KUKA KRL program: EPS_2_251112_SAMH02_A_20250918124114.src

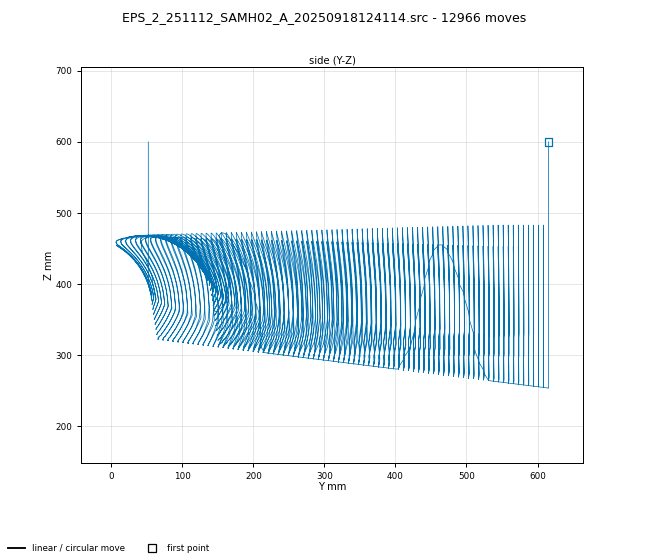
[picture p0: tool path of EPS_2_251112_SAMH02_A_20250918124114.src, 12966 of 12968 moves have a stored position in this frame; points joined in program order, loops and branches not executed]
&ACCESS RVP
&REL 4
&COMMENT QRS 19112012
&PARAM EDITMASK = *
DEF PART()
EXT BAS (BAS_COMMAND :IN,REAL :IN )
INT I
BAS (#INITMOV,0 )

;KUKA QRS Post kuka4.cps  Date:22-06-2017 !

File_ID=2849

QRS_PRE_INIT()

;Init var - Until changes are made in qrs_pre_init
Outlet_Square_prg=0
Inlet_1_Square_prg=0
Inlet_2_Square_prg=0
Inlet_3_Square_prg=0
Inlet_4_Square_prg=0
Inlet_5_Square_prg=0

Outlet_1={X 0.000, Y 541.230, Z 408.000, B 0.000, E1 0.000 }
Inlet_1={X 0.000, Y 543.360, Z 378.000, B 0.000, E1 152.000 }
Outlet_1_type=150
Inlet_1_type=150
;QRS#1=Sidecore dimensions
;QRS#2=150-6" PVC SDR 28
;QRS#3=150-6" PVC SDR 28
;QRS#4=
;QRS#5=
;QRS#6=
;QRS#7=
;QRS#8=
;QRS#9=10-06 PSX
;QRS#10=10-06 PSX
;QRS#11=
;QRS#12=
;QRS#13=
;QRS#14=
;QRS#15=
;QRS#16=1220x127x762 2,5'
;QRS#17=EPS Height
;QRS#18=483
;QRS#19=*
;QRS#20= UPDATED VERSION 22-06-2017
;QRS#21=*
Outlet_Square=070
Inlet_1_Square=070
Inlet_2_Square=0
Inlet_3_Square=0
Inlet_4_Square=0
Inlet_5_Square=0
Mill_Square=1
Outlet_Square_Prg=203
Inlet_1_Square_prg=203

QRS_INIT()

$ADVANCE=5

; T1
PTP {E1 173.623,E2 173.623}
PTP {X 0,Y 615.454,A -85,B 0,C 180,E1 173.623,E2 173.623,E3 0,E4 0,E5 0,E6 0}
QRS_SPEED_INIT()
LIN {X 0,Y 615.454,Z 600,A -85,B 0,C 180,E1 173.623,E2 173.623,E3 0,E4 0,E5 0,E6 0} C_VEL
LIN {X 0,Y 615.454,Z 263.682,A -85,B 0,C 180,E1 173.623,E2 173.623} C_VEL
LIN {X 0,Y 615.454,Z 255.505,A -85,B 0,C 180,E1 173.623,E2 173.623} C_VEL
LIN {X 0,Y 615.45,Z 253.505,A -85,B 0,C 180,E1 173.437,E2 173.437} C_VEL
LIN {X 0,Y 615.491,Z 253.512,A -85,B 0,C 180,E1 170.801,E2 170.801} C_VEL
LIN {X 0,Y 615.491,Z 253.498,A -85,B 0,C 180,E1 168.139,E2 168.139} C_VEL
LIN {X 0,Y 615.456,Z 253.5,A -85,B 0,C 180,E1 165.45,E2 165.45} C_VEL
LIN {X 0,Y 615.458,Z 253.499,A -85,B 0,C 180,E1 163.412,E2 163.412} C_VEL
LIN {X 0,Y 615.459,Z 253.499,A -85,B 0,C 180,E1 161.353,E2 161.353} C_VEL
LIN {X 0,Y 615.459,Z 253.499,A -85,B 0,C 180,E1 159.268,E2 159.268} C_VEL
LIN {X 0,Y 615.458,Z 253.5,A -85,B 0,C 180,E1 157.154,E2 157.154} C_VEL
LIN {X 0,Y 615.456,Z 253.5,A -85,B 0,C 180,E1 155.007,E2 155.007} C_VEL
LIN {X 0,Y 615.454,Z 253.502,A -85,B 0,C 180,E1 152.821,E2 152.821} C_VEL
LIN {X 0,Y 615.475,Z 253.509,A -85,B 0,C 180,E1 150.204,E2 150.204} C_VEL
LIN {X 0,Y 615.489,Z 253.502,A -85,B 0,C 180,E1 147.543,E2 147.543} C_VEL
LIN {X 0,Y 615.496,Z 253.494,A -85,B 0,C 180,E1 145.185,E2 145.185} C_VEL
LIN {X 0,Y 615.469,Z 253.497,A -85,B 0,C 180,E1 142.756,E2 142.756} C_VEL
LIN {X 0,Y 615.456,Z 253.503,A -85,B 0,C 180,E1 140.247,E2 140.247} C_VEL
LIN {X 0,Y 615.486,Z 253.511,A -85,B 0,C 180,E1 137.647,E2 137.647} C_VEL
LIN {X 0,Y 615.461,Z 253.707,A -85,B 0,C 180,E1 135.926,E2 135.926} C_VEL
LIN {X 0,Y 615.484,Z 267.327,A -85,B 0,C 180,E1 133.243,E2 133.243} C_VEL
LIN {X 0,Y 615.489,Z 280.89,A -85,B 0,C 180,E1 130.605,E2 130.605} C_VEL
LIN {X 0,Y 615.477,Z 294.187,A -85,B 0,C 180,E1 128.053,E2 128.053} C_VEL
LIN {X 0,Y 615.497,Z 369.287,A -85,B 0,C 180,E1 127.164,E2 127.164} C_VEL
LIN {X 0,Y 615.489,Z 378.589,A -85,B 0,C 180,E1 126.974,E2 126.974} C_VEL
LIN {X 0,Y 615.487,Z 386.446,A -85,B 0,C 180,E1 126.744,E2 126.744} C_VEL
LIN {X 0,Y 615.49,Z 394.748,A -85,B 0,C 180,E1 126.423,E2 126.423} C_VEL
LIN {X 0,Y 615.494,Z 402.34,A -85,B 0,C 180,E1 126.054,E2 126.054} C_VEL
LIN {X 0,Y 615.478,Z 411.206,A -85,B 0,C 180,E1 125.515,E2 125.515} C_VEL
LIN {X 0,Y 615.492,Z 419.16,A -85,B 0,C 180,E1 124.913,E2 124.913} C_VEL
LIN {X 0,Y 615.496,Z 426.942,A -85,B 0,C 180,E1 124.19,E2 124.19} C_VEL
LIN {X 0,Y 615.494,Z 433.793,A -85,B 0,C 180,E1 123.385,E2 123.385} C_VEL
LIN {X 0,Y 615.499,Z 438.844,A -85,B 0,C 180,E1 122.65,E2 122.65} C_VEL
LIN {X 0,Y 615.493,Z 442.518,A -85,B 0,C 180,E1 122.008,E2 122.008} C_VEL
LIN {X 0,Y 615.489,Z 446.578,A -85,B 0,C 180,E1 121.086,E2 121.086} C_VEL
LIN {X 0,Y 615.499,Z 449.503,A -85,B 0,C 180,E1 120.158,E2 120.158} C_VEL
LIN {X 0,Y 615.49,Z 451.13,A -85,B 0,C 180,E1 119.405,E2 119.405} C_VEL
LIN {X 0,Y 615.494,Z 452.177,A -85,B 0,C 180,E1 118.451,E2 118.451} C_VEL
LIN {X 0,Y 615.491,Z 452.386,A -85,B 0,C 180,E1 117.914,E2 117.914} C_VEL
LIN {X 0,Y 615.487,Z 451.899,A -85,B 0,C 180,E1 117.045,E2 117.045} C_VEL
LIN {X 0,Y 615.489,Z 451.043,A -85,B 0,C 180,E1 116.443,E2 116.443} C_VEL
LIN {X 0,Y 615.492,Z 449.065,A -85,B 0,C 180,E1 115.569,E2 115.569} C_VEL
LIN {X 0,Y 615.493,Z 445.858,A -85,B 0,C 180,E1 114.63,E2 114.63} C_VEL
LIN {X 0,Y 615.496,Z 441.867,A -85,B 0,C 180,E1 113.782,E2 113.782} C_VEL
LIN {X 0,Y 615.494,Z 437.323,A -85,B 0,C 180,E1 113.021,E2 113.021} C_VEL
LIN {X 0,Y 615.498,Z 430.598,A -85,B 0,C 180,E1 112.135,E2 112.135} C_VEL
LIN {X 0,Y 615.499,Z 423.976,A -85,B 0,C 180,E1 111.431,E2 111.431} C_VEL
LIN {X 0,Y 615.482,Z 415.903,A -85,B 0,C 180,E1 110.73,E2 110.73} C_VEL
LIN {X 0,Y 615.489,Z 405.501,A -85,B 0,C 180,E1 110.032,E2 110.032} C_VEL
LIN {X 0,Y 615.482,Z 397.231,A -85,B 0,C 180,E1 109.598,E2 109.598} C_VEL
LIN {X 0,Y 615.474,Z 388.91,A -85,B 0,C 180,E1 109.251,E2 109.251} C_VEL
LIN {X 0,Y 615.487,Z 379.076,A -85,B 0,C 180,E1 108.948,E2 108.948} C_VEL
LIN {X 0,Y 615.486,Z 369.76,A -85,B 0,C 180,E1 108.753,E2 108.753} C_VEL
LIN {X 0,Y 615.48,Z 294.091,A -85,B 0,C 180,E1 107.849,E2 107.849} C_VEL
LIN {X 0,Y 615.493,Z 280.475,A -85,B 0,C 180,E1 105.225,E2 105.225} C_VEL
LIN {X 0,Y 615.475,Z 266.63,A -85,B 0,C 180,E1 102.53,E2 102.53} C_VEL
LIN {X 0,Y 615.472,Z 253.502,A -85,B 0,C 180,E1 99.924,E2 99.924} C_VEL
LIN {X 0,Y 615.484,Z 253.494,A -85,B 0,C 180,E1 97.215,E2 97.215} C_VEL
LIN {X 0,Y 615.48,Z 253.504,A -85,B 0,C 180,E1 94.584,E2 94.584} C_VEL
LIN {X 0,Y 615.483,Z 253.509,A -85,B 0,C 180,E1 91.963,E2 91.963} C_VEL
LIN {X 0,Y 615.472,Z 253.498,A -85,B 0,C 180,E1 89.346,E2 89.346} C_VEL
LIN {X 0,Y 615.489,Z 253.494,A -85,B 0,C 180,E1 86.727,E2 86.727} C_VEL
LIN {X 0,Y 615.485,Z 253.507,A -85,B 0,C 180,E1 84.102,E2 84.102} C_VEL
LIN {X 0,Y 615.475,Z 253.506,A -85,B 0,C 180,E1 81.463,E2 81.463} C_VEL
LIN {X 0,Y 615.479,Z 253.495,A -85,B 0,C 180,E1 78.807,E2 78.807} C_VEL
LIN {X 0,Y 615.48,Z 253.501,A -85,B 0,C 180,E1 76.071,E2 76.071} C_VEL
LIN {X 0,Y 615.484,Z 253.513,A -85,B 0,C 180,E1 73.414,E2 73.414} C_VEL
LIN {X 0,Y 615.469,Z 253.498,A -85,B 0,C 180,E1 70.662,E2 70.662} C_VEL
LIN {X 0,Y 615.484,Z 253.498,A -85,B 0,C 180,E1 67.864,E2 67.864} C_VEL
LIN {X 0,Y 615.481,Z 253.509,A -85,B 0,C 180,E1 65.009,E2 65.009} C_VEL
LIN {X 0,Y 615.474,Z 253.507,A -85,B 0,C 180,E1 62.823,E2 62.823} C_VEL
LIN {X 0,Y 615.47,Z 253.497,A -85,B 0,C 180,E1 60.209,E2 60.209} C_VEL
LIN {X 0,Y 615.488,Z 253.496,A -85,B 0,C 180,E1 57.544,E2 57.544} C_VEL
LIN {X 0,Y 615.484,Z 253.504,A -85,B 0,C 180,E1 55.186,E2 55.186} C_VEL
LIN {X 0,Y 615.49,Z 253.515,A -85,B 0,C 180,E1 52.759,E2 52.759} C_VEL
LIN {X 0,Y 615.464,Z 253.499,A -85,B 0,C 180,E1 49.914,E2 49.914} C_VEL
LIN {X 0,Y 615.472,Z 253.496,A -85,B 0,C 180,E1 47.647,E2 47.647} C_VEL
LIN {X 0,Y 615.486,Z 253.5,A -85,B 0,C 180,E1 44.933,E2 44.933} C_VEL
LIN {X 0,Y 615.494,Z 253.512,A -85,B 0,C 180,E1 42.353,E2 42.353} C_VEL
LIN {X 0,Y 615.461,Z 253.503,A -85,B 0,C 180,E1 39.752,E2 39.752} C_VEL
LIN {X 0,Y 615.486,Z 253.495,A -85,B 0,C 180,E1 36.939,E2 36.939} C_VEL
LIN {X 0,Y 615.491,Z 253.511,A -85,B 0,C 180,E1 34.022,E2 34.022} C_VEL
LIN {X 0,Y 615.468,Z 253.507,A -85,B 0,C 180,E1 31.687,E2 31.687} C_VEL
LIN {X 0,Y 615.459,Z 253.504,A -85,B 0,C 180,E1 29.408,E2 29.408} C_VEL
LIN {X 0,Y 615.46,Z 253.5,A -85,B 0,C 180,E1 27.043,E2 27.043} C_VEL
LIN {X 0,Y 615.491,Z 253.497,A -85,B 0,C 180,E1 24.272,E2 24.272} C_VEL
LIN {X 0,Y 615.476,Z 253.509,A -85,B 0,C 180,E1 21.432,E2 21.432} C_VEL
LIN {X 0,Y 615.474,Z 253.509,A -85,B 0,C 180,E1 19.338,E2 19.338} C_VEL
LIN {X 0,Y 615.46,Z 253.499,A -85,B 0,C 180,E1 16.587,E2 16.587} C_VEL
LIN {X 0,Y 615.492,Z 253.498,A -85,B 0,C 180,E1 13.874,E2 13.874} C_VEL
LIN {X 0,Y 615.486,Z 253.511,A -85,B 0,C 180,E1 11.193,E2 11.193} C_VEL
LIN {X 0,Y 615.452,Z 253.503,A -85,B 0,C 180,E1 8.537,E2 8.537} C_VEL
LIN {X 0,Y 615.48,Z 253.495,A -85,B 0,C 180,E1 5.899,E2 5.899} C_VEL
LIN {X 0,Y 615.491,Z 253.504,A -85,B 0,C 180,E1 3.273,E2 3.273} C_VEL
LIN {X 0,Y 615.47,Z 253.509,A -85,B 0,C 180,E1 0.654,E2 0.654} C_VEL
LIN {X 0,Y 615.451,Z 253.502,A -85,B 0,C 180,E1 -1.963,E2 -1.963} C_VEL
LIN {X 0,Y 615.488,Z 253.495,A -85,B 0,C 180,E1 -4.584,E2 -4.584} C_VEL
LIN {X 0,Y 615.489,Z 253.509,A -85,B 0,C 180,E1 -7.216,E2 -7.216} C_VEL
LIN {X 0,Y 615.458,Z 253.507,A -85,B 0,C 180,E1 -9.863,E2 -9.863} C_VEL
LIN {X 0,Y 615.463,Z 253.508,A -85,B 0,C 180,E1 -11.861,E2 -11.861} C_VEL
LIN {X 0,Y 615.463,Z 253.508,A -85,B 0,C 180,E1 -13.93,E2 -13.93} C_VEL
LIN {X 0,Y 615.447,Z 253.503,A -85,B 0,C 180,E1 -16.424,E2 -16.424} C_VEL
LIN {X 0,Y 615.449,Z 253.502,A -85,B 0,C 180,E1 -18.647,E2 -18.647} C_VEL
LIN {X 0,Y 615.494,Z 253.499,A -85,B 0,C 180,E1 -21.432,E2 -21.432} C_VEL
LIN {X 0,Y 615.464,Z 253.509,A -85,B 0,C 180,E1 -24.273,E2 -24.273} C_VEL
LIN {X 0,Y 615.456,Z 253.508,A -85,B 0,C 180,E1 -26.446,E2 -26.446} C_VEL
LIN {X 0,Y 615.447,Z 253.507,A -85,B 0,C 180,E1 -28.66,E2 -28.66} C_VEL
LIN {X 0,Y 615.444,Z 253.503,A -85,B 0,C 180,E1 -31.082,E2 -31.082} C_VEL
LIN {X 0,Y 615.467,Z 253.499,A -85,B 0,C 180,E1 -33.534,E2 -33.534} C_VEL
LIN {X 0,Y 615.482,Z 253.515,A -85,B 0,C 180,E1 -36.425,E2 -36.425} C_VEL
LIN {X 0,Y 615.445,Z 253.507,A -85,B 0,C 180,E1 -39.059,E2 -39.059} C_VEL
LIN {X 0,Y 615.44,Z 253.504,A -85,B 0,C 180,E1 -41.478,E2 -41.478} C_VEL
LIN {X 0,Y 615.49,Z 253.497,A -85,B 0,C 180,E1 -44.149,E2 -44.149} C_VEL
LIN {X 0,Y 615.475,Z 253.511,A -85,B 0,C 180,E1 -46.954,E2 -46.954} C_VEL
LIN {X 0,Y 615.445,Z 253.507,A -85,B 0,C 180,E1 -49.392,E2 -49.392} C_VEL
LIN {X 0,Y 615.441,Z 253.503,A -85,B 0,C 180,E1 -51.929,E2 -51.929} C_VEL
LIN {X 0,Y 615.469,Z 253.5,A -85,B 0,C 180,E1 -54.384,E2 -54.384} C_VEL
LIN {X 0,Y 615.491,Z 253.501,A -85,B 0,C 180,E1 -56.765,E2 -56.765} C_VEL
LIN {X 0,Y 615.497,Z 253.508,A -85,B 0,C 180,E1 -59.082,E2 -59.082} C_VEL
LIN {X 0,Y 615.464,Z 253.51,A -85,B 0,C 180,E1 -61.554,E2 -61.554} C_VEL
LIN {X 0,Y 615.47,Z 253.511,A -85,B 0,C 180,E1 -63.556,E2 -63.556} C_VEL
LIN {X 0,Y 615.441,Z 253.508,A -85,B 0,C 180,E1 -66.001,E2 -66.001} C_VEL
LIN {X 0,Y 615.455,Z 253.51,A -85,B 0,C 180,E1 -67.863,E2 -67.863} C_VEL
LIN {X 0,Y 615.467,Z 253.526,A -85,B 0,C 180,E1 -68.963,E2 -68.963} C_VEL
LIN {X 0,Y 615.453,Z 271.669,A -85,B 0,C 180,E1 -71.881,E2 -71.881} C_VEL
LIN {X 0,Y 615.482,Z 287.773,A -85,B 0,C 180,E1 -74.435,E2 -74.435} C_VEL
LIN {X 0,Y 615.47,Z 305.003,A -85,B 0,C 180,E1 -77.135,E2 -77.135} C_VEL
LIN {X 0,Y 615.485,Z 322.619,A -85,B 0,C 180,E1 -79.868,E2 -79.868} C_VEL
LIN {X 0,Y 615.472,Z 399.961,A -85,B 0,C 180,E1 -80.801,E2 -80.801} C_VEL
LIN {X 0,Y 615.465,Z 409.713,A -85,B 0,C 180,E1 -81.008,E2 -81.008} C_VEL
LIN {X 0,Y 615.472,Z 420.166,A -85,B 0,C 180,E1 -81.339,E2 -81.339} C_VEL
LIN {X 0,Y 615.498,Z 430.431,A -85,B 0,C 180,E1 -81.794,E2 -81.794} C_VEL
LIN {X 0,Y 615.477,Z 440.204,A -85,B 0,C 180,E1 -82.372,E2 -82.372} C_VEL
LIN {X 0,Y 615.493,Z 447.937,A -85,B 0,C 180,E1 -82.942,E2 -82.942} C_VEL
LIN {X 0,Y 615.497,Z 455.336,A -85,B 0,C 180,E1 -83.608,E2 -83.608} C_VEL
LIN {X 0,Y 615.498,Z 462.739,A -85,B 0,C 180,E1 -84.43,E2 -84.43} C_VEL
LIN {X 0,Y 615.497,Z 468.533,A -85,B 0,C 180,E1 -85.252,E2 -85.252} C_VEL
LIN {X 0,Y 615.494,Z 473.101,A -85,B 0,C 180,E1 -86.072,E2 -86.072} C_VEL
LIN {X 0,Y 615.493,Z 476.069,A -85,B 0,C 180,E1 -86.727,E2 -86.727} C_VEL
LIN {X 0,Y 615.494,Z 478.357,A -85,B 0,C 180,E1 -87.382,E2 -87.382} C_VEL
LIN {X 0,Y 615.499,Z 480.085,A -85,B 0,C 180,E1 -88.037,E2 -88.037} C_VEL
LIN {X 0,Y 615.493,Z 481.33,A -85,B 0,C 180,E1 -88.691,E2 -88.691} C_VEL
LIN {X 0,Y 615.491,Z 482.104,A -85,B 0,C 180,E1 -89.346,E2 -89.346} C_VEL
LIN {X 0,Y 615.491,Z 482.389,A -85,B 0,C 180,E1 -90,E2 -90} C_VEL
LIN {X 0,Y 615.491,Z 482.104,A -85,B 0,C 180,E1 -90.654,E2 -90.654} C_VEL
LIN {X 0,Y 615.493,Z 481.33,A -85,B 0,C 180,E1 -91.309,E2 -91.309} C_VEL
LIN {X 0,Y 615.499,Z 480.085,A -85,B 0,C 180,E1 -91.963,E2 -91.963} C_VEL
LIN {X 0,Y 615.488,Z 477.221,A -85,B 0,C 180,E1 -92.945,E2 -92.945} C_VEL
LIN {X 0,Y 615.492,Z 474.604,A -85,B 0,C 180,E1 -93.601,E2 -93.601} C_VEL
LIN {X 0,Y 615.497,Z 469.483,A -85,B 0,C 180,E1 -94.584,E2 -94.584} C_VEL
LIN {X 0,Y 615.495,Z 463.969,A -85,B 0,C 180,E1 -95.405,E2 -95.405} C_VEL
LIN {X 0,Y 615.498,Z 457.02,A -85,B 0,C 180,E1 -96.227,E2 -96.227} C_VEL
LIN {X 0,Y 615.495,Z 449.86,A -85,B 0,C 180,E1 -96.901,E2 -96.901} C_VEL
LIN {X 0,Y 615.477,Z 442.628,A -85,B 0,C 180,E1 -97.463,E2 -97.463} C_VEL
LIN {X 0,Y 615.495,Z 434.873,A -85,B 0,C 180,E1 -97.958,E2 -97.958} C_VEL
LIN {X 0,Y 615.494,Z 426.92,A -85,B 0,C 180,E1 -98.371,E2 -98.371} C_VEL
LIN {X 0,Y 615.468,Z 417.771,A -85,B 0,C 180,E1 -98.743,E2 -98.743} C_VEL
LIN {X 0,Y 615.465,Z 409.714,A -85,B 0,C 180,E1 -98.992,E2 -98.992} C_VEL
LIN {X 0,Y 615.472,Z 399.963,A -85,B 0,C 180,E1 -99.199,E2 -99.199} C_VEL
LIN {X 0,Y 615.482,Z 322.62,A -85,B 0,C 180,E1 -100.132,E2 -100.132} C_VEL
LIN {X 0,Y 615.47,Z 305.003,A -85,B 0,C 180,E1 -102.865,E2 -102.865} C_VEL
LIN {X 0,Y 615.482,Z 287.773,A -85,B 0,C 180,E1 -105.565,E2 -105.565} C_VEL
LIN {X 0,Y 615.459,Z 270.657,A -85,B 0,C 180,E1 -108.28,E2 -108.28} C_VEL
LIN {X 0,Y 615.464,Z 253.501,A -85,B 0,C 180,E1 -111.059,E2 -111.059} C_VEL
LIN {X 0,Y 615.437,Z 253.504,A -85,B 0,C 180,E1 -113.558,E2 -113.558} C_VEL
LIN {X 0,Y 615.435,Z 253.505,A -85,B 0,C 180,E1 -115.717,E2 -115.717} C_VEL
LIN {X 0,Y 615.435,Z 253.506,A -85,B 0,C 180,E1 -117.917,E2 -117.917} C_VEL
LIN {X 0,Y 615.437,Z 253.507,A -85,B 0,C 180,E1 -120.162,E2 -120.162} C_VEL
LIN {X 0,Y 615.451,Z 253.509,A -85,B 0,C 180,E1 -122.458,E2 -122.458} C_VEL
LIN {X 0,Y 615.48,Z 253.512,A -85,B 0,C 180,E1 -124.814,E2 -124.814} C_VEL
LIN {X 0,Y 615.496,Z 253.505,A -85,B 0,C 180,E1 -127.24,E2 -127.24} C_VEL
LIN {X 0,Y 615.472,Z 253.499,A -85,B 0,C 180,E1 -129.75,E2 -129.75} C_VEL
LIN {X 0,Y 615.439,Z 253.504,A -85,B 0,C 180,E1 -132.356,E2 -132.356} C_VEL
LIN {X 0,Y 615.455,Z 253.509,A -85,B 0,C 180,E1 -134.928,E2 -134.928} C_VEL
LIN {X 0,Y 615.494,Z 253.505,A -85,B 0,C 180,E1 -137.648,E2 -137.648} C_VEL
LIN {X 0,Y 615.462,Z 253.5,A -85,B 0,C 180,E1 -140.248,E2 -140.248} C_VEL
LIN {X 0,Y 615.441,Z 253.504,A -85,B 0,C 180,E1 -142.755,E2 -142.755} C_VEL
LIN {X 0,Y 615.455,Z 253.509,A -85,B 0,C 180,E1 -145.301,E2 -145.301} C_VEL
LIN {X 0,Y 615.485,Z 253.511,A -85,B 0,C 180,E1 -147.667,E2 -147.667} C_VEL
LIN {X 0,Y 615.47,Z 253.499,A -85,B 0,C 180,E1 -150.593,E2 -150.593} C_VEL
LIN {X 0,Y 615.447,Z 253.502,A -85,B 0,C 180,E1 -152.959,E2 -152.959} C_VEL
LIN {X 0,Y 615.451,Z 253.501,A -85,B 0,C 180,E1 -155.007,E2 -155.007} C_VEL
LIN {X 0,Y 615.448,Z 253.502,A -85,B 0,C 180,E1 -157.154,E2 -157.154} C_VEL
LIN {X 0,Y 615.444,Z 253.504,A -85,B 0,C 180,E1 -159.449,E2 -159.449} C_VEL
LIN {X 0,Y 615.469,Z 253.51,A -85,B 0,C 180,E1 -162.043,E2 -162.043} C_VEL
LIN {X 0,Y 615.495,Z 253.5,A -85,B 0,C 180,E1 -164.774,E2 -164.774} C_VEL
LIN {X 0,Y 615.453,Z 253.5,A -85,B 0,C 180,E1 -167.469,E2 -167.469} C_VEL
LIN {X 0,Y 615.458,Z 253.499,A -85,B 0,C 180,E1 -169.473,E2 -169.473} C_VEL
LIN {X 0,Y 615.466,Z 253.498,A -85,B 0,C 180,E1 -171.463,E2 -171.463} C_VEL
LIN {X 0,Y 615.448,Z 253.505,A -85,B 0,C 180,E1 -174.101,E2 -174.101} C_VEL
LIN {X 0,Y 615.486,Z 253.512,A -85,B 0,C 180,E1 -176.727,E2 -176.727} C_VEL
LIN {X 0,Y 615.49,Z 253.499,A -85,B 0,C 180,E1 -179.346,E2 -179.346} C_VEL
LIN {X 0,Y 615.459,Z 253.499,A -85,B 0,C 180,E1 -181.963,E2 -181.963} C_VEL
LIN {X 0,Y 615.453,Z 253.506,A -85,B 0,C 180,E1 -184.585,E2 -184.585} C_VEL
LIN {X 0,Y 615.45,Z 253.505,A -85,B 0,C 180,E1 -186.563,E2 -186.563} C_VEL
LIN {X 0,Y 614.799,Z 253.659,A -85,B 0,C 180,E1 -187.109,E2 -187.109} C_VEL
LIN {X 0,Y 611.984,Z 254.059,A -85,B 0,C 180,E1 -187.996,E2 -187.996} C_VEL
LIN {X 0,Y 609.593,Z 254.377,A -85,B 0,C 180,E1 -188.708,E2 -188.708} C_VEL
LIN {X 0,Y 608.554,Z 254.498,A -85,B 0,C 180,E1 -189.258,E2 -189.258} C_VEL
LIN {X 0,Y 608.463,Z 254.506,A -85,B 0,C 180,E1 -189.444,E2 -189.444} C_VEL
LIN {X 0,Y 608.457,Z 254.5,A -85,B 0,C 180,E1 -192,E2 -192} C_VEL
LIN {X 0,Y 608.45,Z 254.5,A -85,B 0,C 180,E1 -194.721,E2 -194.721} C_VEL
LIN {X 0,Y 608.422,Z 254.503,A -85,B 0,C 180,E1 -196.785,E2 -196.785} C_VEL
LIN {X 0,Y 608.441,Z 254.511,A -85,B 0,C 180,E1 -199.571,E2 -199.571} C_VEL
LIN {X 0,Y 608.45,Z 254.5,A -85,B 0,C 180,E1 -202.478,E2 -202.478} C_VEL
LIN {X 0,Y 608.443,Z 254.501,A -85,B 0,C 180,E1 -204.572,E2 -204.572} C_VEL
LIN {X 0,Y 608.451,Z 254.5,A -85,B 0,C 180,E1 -207.206,E2 -207.206} C_VEL
LIN {X 0,Y 608.462,Z 254.509,A -85,B 0,C 180,E1 -209.974,E2 -209.974} C_VEL
LIN {X 0,Y 608.445,Z 254.5,A -85,B 0,C 180,E1 -212.88,E2 -212.88} C_VEL
LIN {X 0,Y 608.43,Z 254.501,A -85,B 0,C 180,E1 -215.279,E2 -215.279} C_VEL
LIN {X 0,Y 608.453,Z 254.501,A -85,B 0,C 180,E1 -217.748,E2 -217.748} C_VEL
LIN {X 0,Y 608.444,Z 254.511,A -85,B 0,C 180,E1 -220.33,E2 -220.33} C_VEL
LIN {X 0,Y 608.477,Z 254.496,A -85,B 0,C 180,E1 -223.311,E2 -223.311} C_VEL
LIN {X 0,Y 608.445,Z 254.617,A -85,B 0,C 180,E1 -224.02,E2 -224.02} C_VEL
LIN {X 0,Y 608.471,Z 268.075,A -85,B 0,C 180,E1 -226.691,E2 -226.691} C_VEL
LIN {X 0,Y 608.441,Z 282.321,A -85,B 0,C 180,E1 -229.48,E2 -229.48} C_VEL
LIN {X 0,Y 608.437,Z 294.377,A -85,B 0,C 180,E1 -231.818,E2 -231.818} C_VEL
LIN {X 0,Y 608.509,Z 369.385,A -85,B 0,C 180,E1 -232.723,E2 -232.723} C_VEL
LIN {X 0,Y 608.501,Z 378.797,A -85,B 0,C 180,E1 -232.917,E2 -232.917} C_VEL
LIN {X 0,Y 608.505,Z 387.885,A -85,B 0,C 180,E1 -233.193,E2 -233.193} C_VEL
LIN {X 0,Y 608.487,Z 396.712,A -85,B 0,C 180,E1 -233.553,E2 -233.553} C_VEL
LIN {X 0,Y 608.479,Z 405.514,A -85,B 0,C 180,E1 -234.012,E2 -234.012} C_VEL
LIN {X 0,Y 608.446,Z 414.814,A -85,B 0,C 180,E1 -234.622,E2 -234.622} C_VEL
LIN {X 0,Y 608.45,Z 423.03,A -85,B 0,C 180,E1 -235.313,E2 -235.313} C_VEL
LIN {X 0,Y 608.467,Z 429.1,A -85,B 0,C 180,E1 -235.931,E2 -235.931} C_VEL
LIN {X 0,Y 608.436,Z 435.483,A -85,B 0,C 180,E1 -236.725,E2 -236.725} C_VEL
LIN {X 0,Y 608.433,Z 440.417,A -85,B 0,C 180,E1 -237.482,E2 -237.482} C_VEL
LIN {X 0,Y 608.427,Z 444.651,A -85,B 0,C 180,E1 -238.294,E2 -238.294} C_VEL
LIN {X 0,Y 608.421,Z 447.88,A -85,B 0,C 180,E1 -239.093,E2 -239.093} C_VEL
LIN {X 0,Y 608.425,Z 450.622,A -85,B 0,C 180,E1 -240.036,E2 -240.036} C_VEL
LIN {X 0,Y 608.409,Z 452.298,A -85,B 0,C 180,E1 -240.978,E2 -240.978} C_VEL
LIN {X 0,Y 608.438,Z 452.878,A -85,B 0,C 180,E1 -241.734,E2 -241.734} C_VEL
LIN {X 0,Y 608.429,Z 452.666,A -85,B 0,C 180,E1 -242.802,E2 -242.802} C_VEL
LIN {X 0,Y 608.417,Z 450.84,A -85,B 0,C 180,E1 -243.964,E2 -243.964} C_VEL
LIN {X 0,Y 608.429,Z 447.648,A -85,B 0,C 180,E1 -245.064,E2 -245.064} C_VEL
LIN {X 0,Y 608.426,Z 444.364,A -85,B 0,C 180,E1 -245.859,E2 -245.859} C_VEL
LIN {X 0,Y 608.431,Z 439.909,A -85,B 0,C 180,E1 -246.696,E2 -246.696} C_VEL
LIN {X 0,Y 608.458,Z 433.846,A -85,B 0,C 180,E1 -247.595,E2 -247.595} C_VEL
LIN {X 0,Y 608.467,Z 425.99,A -85,B 0,C 180,E1 -248.487,E2 -248.487} C_VEL
LIN {X 0,Y 608.454,Z 419.135,A -85,B 0,C 180,E1 -249.117,E2 -249.117} C_VEL
LIN {X 0,Y 608.457,Z 412.982,A -85,B 0,C 180,E1 -249.594,E2 -249.594} C_VEL
LIN {X 0,Y 608.464,Z 405.503,A -85,B 0,C 180,E1 -250.079,E2 -250.079} C_VEL
LIN {X 0,Y 608.465,Z 397.14,A -85,B 0,C 180,E1 -250.518,E2 -250.518} C_VEL
LIN {X 0,Y 608.488,Z 388.671,A -85,B 0,C 180,E1 -250.87,E2 -250.87} C_VEL
LIN {X 0,Y 608.508,Z 378.997,A -85,B 0,C 180,E1 -251.168,E2 -251.168} C_VEL
LIN {X 0,Y 608.506,Z 369.825,A -85,B 0,C 180,E1 -251.36,E2 -251.36} C_VEL
LIN {X 0,Y 608.447,Z 294.455,A -85,B 0,C 180,E1 -252.263,E2 -252.263} C_VEL
LIN {X 0,Y 608.442,Z 280.641,A -85,B 0,C 180,E1 -254.937,E2 -254.937} C_VEL
LIN {X 0,Y 608.477,Z 268.457,A -85,B 0,C 180,E1 -257.324,E2 -257.324} C_VEL
LIN {X 0,Y 608.468,Z 254.532,A -85,B 0,C 180,E1 -260.086,E2 -260.086} C_VEL
LIN {X 0,Y 608.463,Z 254.497,A -85,B 0,C 180,E1 -262.701,E2 -262.701} C_VEL
LIN {X 0,Y 608.45,Z 254.504,A -85,B 0,C 180,E1 -265.362,E2 -265.362} C_VEL
LIN {X 0,Y 608.453,Z 254.507,A -85,B 0,C 180,E1 -268.014,E2 -268.014} C_VEL
LIN {X 0,Y 608.468,Z 254.498,A -85,B 0,C 180,E1 -270.662,E2 -270.662} C_VEL
LIN {X 0,Y 608.482,Z 254.496,A -85,B 0,C 180,E1 -273.311,E2 -273.311} C_VEL
LIN {X 0,Y 608.457,Z 254.507,A -85,B 0,C 180,E1 -275.967,E2 -275.967} C_VEL
LIN {X 0,Y 608.448,Z 254.503,A -85,B 0,C 180,E1 -278.636,E2 -278.636} C_VEL
LIN {X 0,Y 608.456,Z 254.498,A -85,B 0,C 180,E1 -281.324,E2 -281.324} C_VEL
LIN {X 0,Y 608.47,Z 254.501,A -85,B 0,C 180,E1 -284.037,E2 -284.037} C_VEL
LIN {X 0,Y 608.455,Z 254.505,A -85,B 0,C 180,E1 -286.783,E2 -286.783} C_VEL
LIN {X 0,Y 608.442,Z 254.5,A -85,B 0,C 180,E1 -289.57,E2 -289.57} C_VEL
LIN {X 0,Y 608.477,Z 254.502,A -85,B 0,C 180,E1 -292.405,E2 -292.405} C_VEL
LIN {X 0,Y 608.45,Z 254.507,A -85,B 0,C 180,E1 -294.57,E2 -294.57} C_VEL
LIN {X 0,Y 608.471,Z 254.502,A -85,B 0,C 180,E1 -297.206,E2 -297.206} C_VEL
LIN {X 0,Y 608.461,Z 254.498,A -85,B 0,C 180,E1 -299.97,E2 -299.97} C_VEL
LIN {X 0,Y 608.454,Z 254.506,A -85,B 0,C 180,E1 -302.879,E2 -302.879} C_VEL
LIN {X 0,Y 608.432,Z 254.511,A -85,B 0,C 180,E1 -305.277,E2 -305.277} C_VEL
LIN {X 0,Y 608.457,Z 254.501,A -85,B 0,C 180,E1 -307.746,E2 -307.746} C_VEL
LIN {X 0,Y 608.442,Z 254.5,A -85,B 0,C 180,E1 -310.328,E2 -310.328} C_VEL
LIN {X 0,Y 608.474,Z 254.505,A -85,B 0,C 180,E1 -313.309,E2 -313.309} C_VEL
LIN {X 0,Y 608.454,Z 254.501,A -85,B 0,C 180,E1 -316.129,E2 -316.129} C_VEL
LIN {X 0,Y 608.452,Z 254.499,A -85,B 0,C 180,E1 -318.823,E2 -318.823} C_VEL
LIN {X 0,Y 608.463,Z 254.509,A -85,B 0,C 180,E1 -321.758,E2 -321.758} C_VEL
LIN {X 0,Y 608.466,Z 254.506,A -85,B 0,C 180,E1 -323.95,E2 -323.95} C_VEL
LIN {X 0,Y 608.435,Z 254.505,A -85,B 0,C 180,E1 -326.327,E2 -326.327} C_VEL
LIN {X 0,Y 608.432,Z 254.502,A -85,B 0,C 180,E1 -328.732,E2 -328.732} C_VEL
LIN {X 0,Y 608.471,Z 254.497,A -85,B 0,C 180,E1 -331.377,E2 -331.377} C_VEL
LIN {X 0,Y 608.467,Z 254.507,A -85,B 0,C 180,E1 -334.276,E2 -334.276} C_VEL
LIN {X 0,Y 608.434,Z 254.503,A -85,B 0,C 180,E1 -336.875,E2 -336.875} C_VEL
LIN {X 0,Y 608.451,Z 254.499,A -85,B 0,C 180,E1 -339.321,E2 -339.321} C_VEL
LIN {X 0,Y 608.442,Z 254.502,A -85,B 0,C 180,E1 -341.828,E2 -341.828} C_VEL
LIN {X 0,Y 608.464,Z 254.509,A -85,B 0,C 180,E1 -344.594,E2 -344.594} C_VEL
LIN {X 0,Y 608.452,Z 254.5,A -85,B 0,C 180,E1 -347.322,E2 -347.322} C_VEL
LIN {X 0,Y 608.457,Z 254.499,A -85,B 0,C 180,E1 -350.023,E2 -350.023} C_VEL
LIN {X 0,Y 608.479,Z 254.504,A -85,B 0,C 180,E1 -352.701,E2 -352.701} C_VEL
LIN {X 0,Y 608.428,Z 254.506,A -85,B 0,C 180,E1 -355.362,E2 -355.362} C_VEL
LIN {X 0,Y 608.455,Z 254.504,A -85,B 0,C 180,E1 -357.352,E2 -357.352} C_VEL
LIN {X 0,Y 608.447,Z 254.499,A -85,B 0,C 180,E1 -360,E2 -360} C_VEL
LIN {X 0,Y 608.482,Z 254.497,A -85,B 0,C 180,E1 -362.648,E2 -362.648} C_VEL
LIN {X 0,Y 608.471,Z 254.508,A -85,B 0,C 180,E1 -365.302,E2 -365.302} C_VEL
LIN {X 0,Y 608.45,Z 254.501,A -85,B 0,C 180,E1 -367.967,E2 -367.967} C_VEL
LIN {X 0,Y 608.447,Z 254.5,A -85,B 0,C 180,E1 -370.65,E2 -370.65} C_VEL
LIN {X 0,Y 608.462,Z 254.505,A -85,B 0,C 180,E1 -373.356,E2 -373.356} C_VEL
LIN {X 0,Y 608.437,Z 254.505,A -85,B 0,C 180,E1 -376.094,E2 -376.094} C_VEL
LIN {X 0,Y 608.436,Z 254.501,A -85,B 0,C 180,E1 -378.87,E2 -378.87} C_VEL
LIN {X 0,Y 608.466,Z 254.505,A -85,B 0,C 180,E1 -381.692,E2 -381.692} C_VEL
LIN {X 0,Y 608.428,Z 254.504,A -85,B 0,C 180,E1 -384.572,E2 -384.572} C_VEL
LIN {X 0,Y 608.451,Z 254.499,A -85,B 0,C 180,E1 -387.206,E2 -387.206} C_VEL
LIN {X 0,Y 608.474,Z 254.504,A -85,B 0,C 180,E1 -389.976,E2 -389.976} C_VEL
LIN {X 0,Y 608.433,Z 254.503,A -85,B 0,C 180,E1 -392.881,E2 -392.881} C_VEL
LIN {X 0,Y 608.417,Z 254.503,A -85,B 0,C 180,E1 -395.279,E2 -395.279} C_VEL
LIN {X 0,Y 608.455,Z 254.499,A -85,B 0,C 180,E1 -397.747,E2 -397.747} C_VEL
LIN {X 0,Y 608.473,Z 254.504,A -85,B 0,C 180,E1 -400.333,E2 -400.333} C_VEL
LIN {X 0,Y 608.425,Z 254.508,A -85,B 0,C 180,E1 -402.962,E2 -402.962} C_VEL
LIN {X 0,Y 608.427,Z 254.505,A -85,B 0,C 180,E1 -405.203,E2 -405.203} C_VEL
LIN {X 0,Y 608.436,Z 254.507,A -85,B 0,C 180,E1 -407.04,E2 -407.04} C_VEL
LIN {X 0,Y 608.41,Z 254.504,A -85,B 0,C 180,E1 -409.695,E2 -409.695} C_VEL
LIN {X 0,Y 608.445,Z 254.501,A -85,B 0,C 180,E1 -412.253,E2 -412.253} C_VEL
LIN {X 0,Y 608.445,Z 254.511,A -85,B 0,C 180,E1 -415.095,E2 -415.095} C_VEL
LIN {X 0,Y 608.428,Z 254.502,A -85,B 0,C 180,E1 -417.904,E2 -417.904} C_VEL
LIN {X 0,Y 608.423,Z 254.502,A -85,B 0,C 180,E1 -420.219,E2 -420.219} C_VEL
LIN {X 0,Y 608.458,Z 254.501,A -85,B 0,C 180,E1 -422.797,E2 -422.797} C_VEL
LIN {X 0,Y 608.445,Z 254.504,A -85,B 0,C 180,E1 -425.854,E2 -425.854} C_VEL
LIN {X 0,Y 608.429,Z 254.503,A -85,B 0,C 180,E1 -428.308,E2 -428.308} C_VEL
LIN {X 0,Y 608.456,Z 254.629,A -85,B 0,C 180,E1 -428.886,E2 -428.886} C_VEL
LIN {X 0,Y 608.48,Z 271.013,A -85,B 0,C 180,E1 -431.551,E2 -431.551} C_VEL
LIN {X 0,Y 608.5,Z 287.882,A -85,B 0,C 180,E1 -434.252,E2 -434.252} C_VEL
LIN {X 0,Y 608.443,Z 305.184,A -85,B 0,C 180,E1 -436.983,E2 -436.983} C_VEL
LIN {X 0,Y 608.471,Z 322.892,A -85,B 0,C 180,E1 -439.75,E2 -439.75} C_VEL
LIN {X 0,Y 608.495,Z 400.46,A -85,B 0,C 180,E1 -440.695,E2 -440.695} C_VEL
LIN {X 0,Y 608.464,Z 410.085,A -85,B 0,C 180,E1 -440.904,E2 -440.904} C_VEL
LIN {X 0,Y 608.479,Z 421.623,A -85,B 0,C 180,E1 -441.281,E2 -441.281} C_VEL
LIN {X 0,Y 608.479,Z 432.237,A -85,B 0,C 180,E1 -441.783,E2 -441.783} C_VEL
LIN {X 0,Y 608.458,Z 440.545,A -85,B 0,C 180,E1 -442.284,E2 -442.284} C_VEL
LIN {X 0,Y 608.459,Z 448.403,A -85,B 0,C 180,E1 -442.868,E2 -442.868} C_VEL
LIN {X 0,Y 608.466,Z 455.358,A -85,B 0,C 180,E1 -443.496,E2 -443.496} C_VEL
LIN {X 0,Y 608.469,Z 463.192,A -85,B 0,C 180,E1 -444.366,E2 -444.366} C_VEL
LIN {X 0,Y 608.448,Z 469.028,A -85,B 0,C 180,E1 -445.196,E2 -445.196} C_VEL
LIN {X 0,Y 608.432,Z 473.631,A -85,B 0,C 180,E1 -446.026,E2 -446.026} C_VEL
LIN {X 0,Y 608.425,Z 476.622,A -85,B 0,C 180,E1 -446.689,E2 -446.689} C_VEL
LIN {X 0,Y 608.423,Z 478.931,A -85,B 0,C 180,E1 -447.352,E2 -447.352} C_VEL
LIN {X 0,Y 608.443,Z 480.678,A -85,B 0,C 180,E1 -448.014,E2 -448.014} C_VEL
LIN {X 0,Y 608.446,Z 481.934,A -85,B 0,C 180,E1 -448.676,E2 -448.676} C_VEL
LIN {X 0,Y 608.434,Z 482.714,A -85,B 0,C 180,E1 -449.338,E2 -449.338} C_VEL
LIN {X 0,Y 608.431,Z 483,A -85,B 0,C 180,E1 -450,E2 -450} C_VEL
LIN {X 0,Y 608.434,Z 482.714,A -85,B 0,C 180,E1 -450.662,E2 -450.662} C_VEL
LIN {X 0,Y 608.446,Z 481.934,A -85,B 0,C 180,E1 -451.324,E2 -451.324} C_VEL
LIN {X 0,Y 608.443,Z 480.678,A -85,B 0,C 180,E1 -451.986,E2 -451.986} C_VEL
LIN {X 0,Y 608.444,Z 477.786,A -85,B 0,C 180,E1 -452.979,E2 -452.979} C_VEL
LIN {X 0,Y 608.446,Z 475.147,A -85,B 0,C 180,E1 -453.642,E2 -453.642} C_VEL
LIN {X 0,Y 608.447,Z 469.986,A -85,B 0,C 180,E1 -454.638,E2 -454.638} C_VEL
LIN {X 0,Y 608.46,Z 464.431,A -85,B 0,C 180,E1 -455.468,E2 -455.468} C_VEL
LIN {X 0,Y 608.455,Z 456.67,A -85,B 0,C 180,E1 -456.376,E2 -456.376} C_VEL
LIN {X 0,Y 608.452,Z 449.418,A -85,B 0,C 180,E1 -457.049,E2 -457.049} C_VEL
LIN {X 0,Y 608.458,Z 441.763,A -85,B 0,C 180,E1 -457.633,E2 -457.633} C_VEL
LIN {X 0,Y 608.497,Z 433.724,A -85,B 0,C 180,E1 -458.134,E2 -458.134} C_VEL
LIN {X 0,Y 608.483,Z 425.395,A -85,B 0,C 180,E1 -458.552,E2 -458.552} C_VEL
LIN {X 0,Y 608.459,Z 416.896,A -85,B 0,C 180,E1 -458.887,E2 -458.887} C_VEL
LIN {X 0,Y 608.491,Z 407.596,A -85,B 0,C 180,E1 -459.159,E2 -459.159} C_VEL
LIN {X 0,Y 608.483,Z 397.864,A -85,B 0,C 180,E1 -459.347,E2 -459.347} C_VEL
LIN {X 0,Y 608.449,Z 322.892,A -85,B 0,C 180,E1 -460.25,E2 -460.25} C_VEL
LIN {X 0,Y 608.443,Z 304.103,A -85,B 0,C 180,E1 -463.186,E2 -463.186} C_VEL
LIN {X 0,Y 608.492,Z 286.8,A -85,B 0,C 180,E1 -465.92,E2 -465.92} C_VEL
LIN {X 0,Y 608.51,Z 269.285,A -85,B 0,C 180,E1 -468.727,E2 -468.727} C_VEL
LIN {X 0,Y 608.428,Z 254.504,A -85,B 0,C 180,E1 -471.137,E2 -471.137} C_VEL
LIN {X 0,Y 608.433,Z 254.503,A -85,B 0,C 180,E1 -473.124,E2 -473.124} C_VEL
LIN {X 0,Y 608.431,Z 254.501,A -85,B 0,C 180,E1 -475.713,E2 -475.713} C_VEL
LIN {X 0,Y 608.416,Z 254.507,A -85,B 0,C 180,E1 -478.267,E2 -478.267} C_VEL
LIN {X 0,Y 608.436,Z 254.508,A -85,B 0,C 180,E1 -480.546,E2 -480.546} C_VEL
LIN {X 0,Y 608.447,Z 254.512,A -85,B 0,C 180,E1 -482.879,E2 -482.879} C_VEL
LIN {X 0,Y 608.431,Z 254.507,A -85,B 0,C 180,E1 -485.277,E2 -485.277} C_VEL
LIN {X 0,Y 608.445,Z 254.501,A -85,B 0,C 180,E1 -487.747,E2 -487.747} C_VEL
LIN {X 0,Y 608.424,Z 254.503,A -85,B 0,C 180,E1 -490.326,E2 -490.326} C_VEL
LIN {X 0,Y 608.435,Z 254.507,A -85,B 0,C 180,E1 -492.96,E2 -492.96} C_VEL
LIN {X 0,Y 608.456,Z 254.503,A -85,B 0,C 180,E1 -495.734,E2 -495.734} C_VEL
LIN {X 0,Y 608.471,Z 254.499,A -85,B 0,C 180,E1 -497.94,E2 -497.94} C_VEL
LIN {X 0,Y 608.415,Z 254.503,A -85,B 0,C 180,E1 -500.556,E2 -500.556} C_VEL
LIN {X 0,Y 608.418,Z 254.506,A -85,B 0,C 180,E1 -503.082,E2 -503.082} C_VEL
LIN {X 0,Y 608.451,Z 254.507,A -85,B 0,C 180,E1 -505.53,E2 -505.53} C_VEL
LIN {X 0,Y 608.465,Z 254.507,A -85,B 0,C 180,E1 -507.906,E2 -507.906} C_VEL
LIN {X 0,Y 608.477,Z 254.501,A -85,B 0,C 180,E1 -510.221,E2 -510.221} C_VEL
LIN {X 0,Y 608.45,Z 254.499,A -85,B 0,C 180,E1 -512.795,E2 -512.795} C_VEL
LIN {X 0,Y 608.426,Z 254.504,A -85,B 0,C 180,E1 -515.428,E2 -515.428} C_VEL
LIN {X 0,Y 608.464,Z 254.506,A -85,B 0,C 180,E1 -518.308,E2 -518.308} C_VEL
LIN {X 0,Y 608.441,Z 254.5,A -85,B 0,C 180,E1 -521.287,E2 -521.287} C_VEL
LIN {X 0,Y 608.434,Z 254.505,A -85,B 0,C 180,E1 -523.906,E2 -523.906} C_VEL
LIN {X 0,Y 608.461,Z 254.506,A -85,B 0,C 180,E1 -526.644,E2 -526.644} C_VEL
LIN {X 0,Y 608.446,Z 254.5,A -85,B 0,C 180,E1 -529.35,E2 -529.35} C_VEL
LIN {X 0,Y 608.447,Z 254.501,A -85,B 0,C 180,E1 -532.033,E2 -532.033} C_VEL
LIN {X 0,Y 608.468,Z 254.508,A -85,B 0,C 180,E1 -534.698,E2 -534.698} C_VEL
LIN {X 0,Y 608.482,Z 254.498,A -85,B 0,C 180,E1 -537.352,E2 -537.352} C_VEL
LIN {X 0,Y 608.445,Z 254.499,A -85,B 0,C 180,E1 -540,E2 -540} C_VEL
LIN {X 0,Y 608.451,Z 254.503,A -85,B 0,C 180,E1 -542.648,E2 -542.648} C_VEL
LIN {X 0,Y 608.468,Z 254.505,A -85,B 0,C 180,E1 -545.302,E2 -545.302} C_VEL
LIN {X 0,Y 608.468,Z 254.497,A -85,B 0,C 180,E1 -547.967,E2 -547.967} C_VEL
LIN {X 0,Y 608.463,Z 254.506,A -85,B 0,C 180,E1 -549.444,E2 -549.444} C_VEL
LIN {X 0,Y 607.781,Z 254.585,A -85,B 0,C 180,E1 -549.997,E2 -549.997} C_VEL
LIN {X 0,Y 604.925,Z 254.942,A -85,B 0,C 180,E1 -550.893,E2 -550.893} C_VEL
LIN {X 0,Y 602.52,Z 255.244,A -85,B 0,C 180,E1 -551.615,E2 -551.615} C_VEL
LIN {X 0,Y 601.483,Z 255.368,A -85,B 0,C 180,E1 -552.171,E2 -552.171} C_VEL
LIN {X 0,Y 601.395,Z 255.377,A -85,B 0,C 180,E1 -552.36,E2 -552.36} C_VEL
LIN {X 0,Y 601.41,Z 255.378,A -85,B 0,C 180,E1 -554.898,E2 -554.898} C_VEL
LIN {X 0,Y 601.397,Z 255.38,A -85,B 0,C 180,E1 -556.987,E2 -556.987} C_VEL
LIN {X 0,Y 601.397,Z 255.386,A -85,B 0,C 180,E1 -559.81,E2 -559.81} C_VEL
LIN {X 0,Y 601.399,Z 255.378,A -85,B 0,C 180,E1 -562.684,E2 -562.684} C_VEL
LIN {X 0,Y 601.387,Z 255.379,A -85,B 0,C 180,E1 -564.879,E2 -564.879} C_VEL
LIN {X 0,Y 601.395,Z 255.38,A -85,B 0,C 180,E1 -567.362,E2 -567.362} C_VEL
LIN {X 0,Y 601.437,Z 255.382,A -85,B 0,C 180,E1 -570.164,E2 -570.164} C_VEL
LIN {X 0,Y 601.416,Z 255.377,A -85,B 0,C 180,E1 -572.717,E2 -572.717} C_VEL
LIN {X 0,Y 601.406,Z 255.376,A -85,B 0,C 180,E1 -575.116,E2 -575.116} C_VEL
LIN {X 0,Y 601.424,Z 255.375,A -85,B 0,C 180,E1 -577.42,E2 -577.42} C_VEL
LIN {X 0,Y 601.4,Z 255.382,A -85,B 0,C 180,E1 -579.996,E2 -579.996} C_VEL
LIN {X 0,Y 601.408,Z 255.385,A -85,B 0,C 180,E1 -582.671,E2 -582.671} C_VEL
LIN {X 0,Y 601.425,Z 255.557,A -85,B 0,C 180,E1 -583.992,E2 -583.992} C_VEL
LIN {X 0,Y 601.428,Z 268.824,A -85,B 0,C 180,E1 -586.656,E2 -586.656} C_VEL
LIN {X 0,Y 601.394,Z 282.821,A -85,B 0,C 180,E1 -589.429,E2 -589.429} C_VEL
LIN {X 0,Y 601.377,Z 294.376,A -85,B 0,C 180,E1 -591.696,E2 -591.696} C_VEL
LIN {X 0,Y 601.507,Z 369.143,A -85,B 0,C 180,E1 -592.609,E2 -592.609} C_VEL
LIN {X 0,Y 601.479,Z 378.784,A -85,B 0,C 180,E1 -592.809,E2 -592.809} C_VEL
LIN {X 0,Y 601.476,Z 388.492,A -85,B 0,C 180,E1 -593.11,E2 -593.11} C_VEL
LIN {X 0,Y 601.458,Z 398.068,A -85,B 0,C 180,E1 -593.515,E2 -593.515} C_VEL
LIN {X 0,Y 601.41,Z 409.396,A -85,B 0,C 180,E1 -594.158,E2 -594.158} C_VEL
LIN {X 0,Y 601.395,Z 417.689,A -85,B 0,C 180,E1 -594.769,E2 -594.769} C_VEL
LIN {X 0,Y 601.412,Z 424.455,A -85,B 0,C 180,E1 -595.375,E2 -595.375} C_VEL
LIN {X 0,Y 601.376,Z 430.908,A -85,B 0,C 180,E1 -596.073,E2 -596.073} C_VEL
LIN {X 0,Y 601.372,Z 436.793,A -85,B 0,C 180,E1 -596.85,E2 -596.85} C_VEL
LIN {X 0,Y 601.344,Z 442.938,A -85,B 0,C 180,E1 -597.876,E2 -597.876} C_VEL
LIN {X 0,Y 601.35,Z 446.036,A -85,B 0,C 180,E1 -598.557,E2 -598.557} C_VEL
LIN {X 0,Y 601.352,Z 449.198,A -85,B 0,C 180,E1 -599.445,E2 -599.445} C_VEL
LIN {X 0,Y 601.336,Z 451.791,A -85,B 0,C 180,E1 -600.603,E2 -600.603} C_VEL
LIN {X 0,Y 601.325,Z 452.71,A -85,B 0,C 180,E1 -601.369,E2 -601.369} C_VEL
LIN {X 0,Y 601.332,Z 452.984,A -85,B 0,C 180,E1 -602.129,E2 -602.129} C_VEL
LIN {X 0,Y 601.326,Z 452.61,A -85,B 0,C 180,E1 -602.884,E2 -602.884} C_VEL
LIN {X 0,Y 601.311,Z 451.583,A -85,B 0,C 180,E1 -603.633,E2 -603.633} C_VEL
LIN {X 0,Y 601.335,Z 448.846,A -85,B 0,C 180,E1 -604.75,E2 -604.75} C_VEL
LIN {X 0,Y 601.325,Z 445.143,A -85,B 0,C 180,E1 -605.731,E2 -605.731} C_VEL
LIN {X 0,Y 601.363,Z 441.878,A -85,B 0,C 180,E1 -606.406,E2 -606.406} C_VEL
LIN {X 0,Y 601.36,Z 437.536,A -85,B 0,C 180,E1 -607.134,E2 -607.134} C_VEL
LIN {X 0,Y 601.373,Z 432.23,A -85,B 0,C 180,E1 -607.861,E2 -607.861} C_VEL
LIN {X 0,Y 601.412,Z 425.799,A -85,B 0,C 180,E1 -608.582,E2 -608.582} C_VEL
LIN {X 0,Y 601.4,Z 418.107,A -85,B 0,C 180,E1 -609.286,E2 -609.286} C_VEL
LIN {X 0,Y 601.418,Z 410.79,A -85,B 0,C 180,E1 -609.835,E2 -609.835} C_VEL
LIN {X 0,Y 601.427,Z 402.057,A -85,B 0,C 180,E1 -610.37,E2 -610.37} C_VEL
LIN {X 0,Y 601.479,Z 390.647,A -85,B 0,C 180,E1 -610.904,E2 -610.904} C_VEL
LIN {X 0,Y 601.49,Z 379.692,A -85,B 0,C 180,E1 -611.258,E2 -611.258} C_VEL
LIN {X 0,Y 601.511,Z 370.659,A -85,B 0,C 180,E1 -611.456,E2 -611.456} C_VEL
LIN {X 0,Y 601.499,Z 327.876,A -85,B 0,C 180,E1 -611.986,E2 -611.986} C_VEL
LIN {X 0,Y 601.417,Z 294.916,A -85,B 0,C 180,E1 -612.379,E2 -612.379} C_VEL
LIN {X 0,Y 601.387,Z 294.344,A -85,B 0,C 180,E1 -612.4,E2 -612.4} C_VEL
LIN {X 0,Y 601.373,Z 280.585,A -85,B 0,C 180,E1 -615.102,E2 -615.102} C_VEL
LIN {X 0,Y 601.433,Z 268.413,A -85,B 0,C 180,E1 -617.516,E2 -617.516} C_VEL
LIN {X 0,Y 601.415,Z 255.379,A -85,B 0,C 180,E1 -620.16,E2 -620.16} C_VEL
LIN {X 0,Y 601.44,Z 255.372,A -85,B 0,C 180,E1 -622.615,E2 -622.615} C_VEL
LIN {X 0,Y 601.419,Z 255.379,A -85,B 0,C 180,E1 -625.308,E2 -625.308} C_VEL
LIN {X 0,Y 601.423,Z 255.383,A -85,B 0,C 180,E1 -627.991,E2 -627.991} C_VEL
LIN {X 0,Y 601.441,Z 255.373,A -85,B 0,C 180,E1 -630.67,E2 -630.67} C_VEL
LIN {X 0,Y 601.433,Z 255.374,A -85,B 0,C 180,E1 -633.349,E2 -633.349} C_VEL
LIN {X 0,Y 601.407,Z 255.386,A -85,B 0,C 180,E1 -636.037,E2 -636.037} C_VEL
LIN {X 0,Y 601.437,Z 255.382,A -85,B 0,C 180,E1 -638.061,E2 -638.061} C_VEL
LIN {X 0,Y 601.42,Z 255.376,A -85,B 0,C 180,E1 -641.009,E2 -641.009} C_VEL
LIN {X 0,Y 601.411,Z 255.376,A -85,B 0,C 180,E1 -643.516,E2 -643.516} C_VEL
LIN {X 0,Y 601.439,Z 255.38,A -85,B 0,C 180,E1 -646.286,E2 -646.286} C_VEL
LIN {X 0,Y 601.415,Z 255.378,A -85,B 0,C 180,E1 -649.098,E2 -649.098} C_VEL
LIN {X 0,Y 601.402,Z 255.379,A -85,B 0,C 180,E1 -651.239,E2 -651.239} C_VEL
LIN {X 0,Y 601.458,Z 255.372,A -85,B 0,C 180,E1 -654.14,E2 -654.14} C_VEL
LIN {X 0,Y 601.445,Z 255.379,A -85,B 0,C 180,E1 -657.111,E2 -657.111} C_VEL
LIN {X 0,Y 601.409,Z 255.38,A -85,B 0,C 180,E1 -659.393,E2 -659.393} C_VEL
LIN {X 0,Y 601.399,Z 255.379,A -85,B 0,C 180,E1 -661.726,E2 -661.726} C_VEL
LIN {X 0,Y 601.415,Z 255.375,A -85,B 0,C 180,E1 -664.118,E2 -664.118} C_VEL
LIN {X 0,Y 601.432,Z 255.382,A -85,B 0,C 180,E1 -667.381,E2 -667.381} C_VEL
LIN {X 0,Y 601.395,Z 255.379,A -85,B 0,C 180,E1 -669.995,E2 -669.995} C_VEL
LIN {X 0,Y 601.405,Z 255.377,A -85,B 0,C 180,E1 -672.669,E2 -672.669} C_VEL
LIN {X 0,Y 601.419,Z 255.386,A -85,B 0,C 180,E1 -675.481,E2 -675.481} C_VEL
LIN {X 0,Y 601.414,Z 255.376,A -85,B 0,C 180,E1 -678.406,E2 -678.406} C_VEL
LIN {X 0,Y 601.43,Z 255.374,A -85,B 0,C 180,E1 -680.875,E2 -680.875} C_VEL
LIN {X 0,Y 601.435,Z 255.383,A -85,B 0,C 180,E1 -683.733,E2 -683.733} C_VEL
LIN {X 0,Y 601.423,Z 255.383,A -85,B 0,C 180,E1 -686.063,E2 -686.063} C_VEL
LIN {X 0,Y 601.407,Z 255.379,A -85,B 0,C 180,E1 -688.545,E2 -688.545} C_VEL
LIN {X 0,Y 601.432,Z 255.373,A -85,B 0,C 180,E1 -691.209,E2 -691.209} C_VEL
LIN {X 0,Y 601.398,Z 255.38,A -85,B 0,C 180,E1 -693.636,E2 -693.636} C_VEL
LIN {X 0,Y 601.41,Z 255.382,A -85,B 0,C 180,E1 -696.589,E2 -696.589} C_VEL
LIN {X 0,Y 601.419,Z 255.375,A -85,B 0,C 180,E1 -699.478,E2 -699.478} C_VEL
LIN {X 0,Y 601.389,Z 255.387,A -85,B 0,C 180,E1 -702.311,E2 -702.311} C_VEL
LIN {X 0,Y 601.414,Z 255.384,A -85,B 0,C 180,E1 -704.409,E2 -704.409} C_VEL
LIN {X 0,Y 601.402,Z 255.38,A -85,B 0,C 180,E1 -707.171,E2 -707.171} C_VEL
LIN {X 0,Y 601.428,Z 255.374,A -85,B 0,C 180,E1 -709.905,E2 -709.905} C_VEL
LIN {X 0,Y 601.446,Z 255.379,A -85,B 0,C 180,E1 -712.615,E2 -712.615} C_VEL
LIN {X 0,Y 601.4,Z 255.382,A -85,B 0,C 180,E1 -715.308,E2 -715.308} C_VEL
LIN {X 0,Y 601.402,Z 255.377,A -85,B 0,C 180,E1 -717.991,E2 -717.991} C_VEL
LIN {X 0,Y 601.451,Z 255.374,A -85,B 0,C 180,E1 -720.669,E2 -720.669} C_VEL
LIN {X 0,Y 601.425,Z 255.383,A -85,B 0,C 180,E1 -723.349,E2 -723.349} C_VEL
LIN {X 0,Y 601.383,Z 255.38,A -85,B 0,C 180,E1 -726.037,E2 -726.037} C_VEL
LIN {X 0,Y 601.416,Z 255.377,A -85,B 0,C 180,E1 -728.061,E2 -728.061} C_VEL
LIN {X 0,Y 601.459,Z 255.373,A -85,B 0,C 180,E1 -731.038,E2 -731.038} C_VEL
LIN {X 0,Y 601.404,Z 255.38,A -85,B 0,C 180,E1 -734.092,E2 -734.092} C_VEL
LIN {X 0,Y 601.401,Z 255.378,A -85,B 0,C 180,E1 -736.987,E2 -736.987} C_VEL
LIN {X 0,Y 601.396,Z 255.39,A -85,B 0,C 180,E1 -739.81,E2 -739.81} C_VEL
LIN {X 0,Y 601.397,Z 255.378,A -85,B 0,C 180,E1 -742.684,E2 -742.684} C_VEL
LIN {X 0,Y 601.384,Z 255.379,A -85,B 0,C 180,E1 -744.879,E2 -744.879} C_VEL
LIN {X 0,Y 601.408,Z 255.384,A -85,B 0,C 180,E1 -747.868,E2 -747.868} C_VEL
LIN {X 0,Y 601.437,Z 255.385,A -85,B 0,C 180,E1 -750.163,E2 -750.163} C_VEL
LIN {X 0,Y 601.41,Z 255.376,A -85,B 0,C 180,E1 -753.315,E2 -753.315} C_VEL
LIN {X 0,Y 601.432,Z 255.383,A -85,B 0,C 180,E1 -756.267,E2 -756.267} C_VEL
LIN {X 0,Y 601.386,Z 255.381,A -85,B 0,C 180,E1 -759.128,E2 -759.128} C_VEL
LIN {X 0,Y 601.413,Z 255.376,A -85,B 0,C 180,E1 -761.766,E2 -761.766} C_VEL
LIN {X 0,Y 601.416,Z 255.384,A -85,B 0,C 180,E1 -764.536,E2 -764.536} C_VEL
LIN {X 0,Y 601.442,Z 255.378,A -85,B 0,C 180,E1 -766.426,E2 -766.426} C_VEL
LIN {X 0,Y 601.398,Z 255.38,A -85,B 0,C 180,E1 -769.429,E2 -769.429} C_VEL
LIN {X 0,Y 601.385,Z 255.38,A -85,B 0,C 180,E1 -771.731,E2 -771.731} C_VEL
LIN {X 0,Y 601.372,Z 255.381,A -85,B 0,C 180,E1 -774.246,E2 -774.246} C_VEL
LIN {X 0,Y 601.408,Z 255.38,A -85,B 0,C 180,E1 -776.686,E2 -776.686} C_VEL
LIN {X 0,Y 601.4,Z 255.386,A -85,B 0,C 180,E1 -779.058,E2 -779.058} C_VEL
LIN {X 0,Y 601.423,Z 255.385,A -85,B 0,C 180,E1 -781.374,E2 -781.374} C_VEL
LIN {X 0,Y 601.388,Z 255.385,A -85,B 0,C 180,E1 -783.636,E2 -783.636} C_VEL
LIN {X 0,Y 601.425,Z 255.378,A -85,B 0,C 180,E1 -785.859,E2 -785.859} C_VEL
LIN {X 0,Y 601.416,Z 255.44,A -85,B 0,C 180,E1 -788.762,E2 -788.762} C_VEL
LIN {X 0,Y 601.524,Z 268.416,A -85,B 0,C 180,E1 -790.905,E2 -790.905} C_VEL
LIN {X 0,Y 601.456,Z 285.719,A -85,B 0,C 180,E1 -793.714,E2 -793.714} C_VEL
LIN {X 0,Y 601.403,Z 301.187,A -85,B 0,C 180,E1 -796.192,E2 -796.192} C_VEL
LIN {X 0,Y 601.401,Z 317.877,A -85,B 0,C 180,E1 -798.838,E2 -798.838} C_VEL
LIN {X 0,Y 601.407,Z 322.892,A -85,B 0,C 180,E1 -799.628,E2 -799.628} C_VEL
LIN {X 0,Y 601.524,Z 387.927,A -85,B 0,C 180,E1 -800.416,E2 -800.416} C_VEL
LIN {X 0,Y 601.491,Z 404.182,A -85,B 0,C 180,E1 -800.649,E2 -800.649} C_VEL
LIN {X 0,Y 601.457,Z 415.693,A -85,B 0,C 180,E1 -800.967,E2 -800.967} C_VEL
LIN {X 0,Y 601.468,Z 423.542,A -85,B 0,C 180,E1 -801.263,E2 -801.263} C_VEL
LIN {X 0,Y 601.448,Z 432.24,A -85,B 0,C 180,E1 -801.686,E2 -801.686} C_VEL
LIN {X 0,Y 601.402,Z 440.547,A -85,B 0,C 180,E1 -802.192,E2 -802.192} C_VEL
LIN {X 0,Y 601.409,Z 448.404,A -85,B 0,C 180,E1 -802.783,E2 -802.783} C_VEL
LIN {X 0,Y 601.411,Z 455.598,A -85,B 0,C 180,E1 -803.443,E2 -803.443} C_VEL
LIN {X 0,Y 601.391,Z 463.192,A -85,B 0,C 180,E1 -804.299,E2 -804.299} C_VEL
LIN {X 0,Y 601.38,Z 469.028,A -85,B 0,C 180,E1 -805.14,E2 -805.14} C_VEL
LIN {X 0,Y 601.344,Z 473.631,A -85,B 0,C 180,E1 -805.979,E2 -805.979} C_VEL
LIN {X 0,Y 601.344,Z 476.622,A -85,B 0,C 180,E1 -806.65,E2 -806.65} C_VEL
LIN {X 0,Y 601.326,Z 478.932,A -85,B 0,C 180,E1 -807.321,E2 -807.321} C_VEL
LIN {X 0,Y 601.342,Z 480.679,A -85,B 0,C 180,E1 -807.991,E2 -807.991} C_VEL
LIN {X 0,Y 601.345,Z 481.934,A -85,B 0,C 180,E1 -808.661,E2 -808.661} C_VEL
LIN {X 0,Y 601.335,Z 482.713,A -85,B 0,C 180,E1 -809.33,E2 -809.33} C_VEL
LIN {X 0,Y 601.332,Z 483,A -85,B 0,C 180,E1 -810,E2 -810} C_VEL
LIN {X 0,Y 601.335,Z 482.713,A -85,B 0,C 180,E1 -810.67,E2 -810.67} C_VEL
LIN {X 0,Y 601.345,Z 481.934,A -85,B 0,C 180,E1 -811.339,E2 -811.339} C_VEL
LIN {X 0,Y 601.342,Z 480.679,A -85,B 0,C 180,E1 -812.009,E2 -812.009} C_VEL
LIN {X 0,Y 601.343,Z 477.787,A -85,B 0,C 180,E1 -813.015,E2 -813.015} C_VEL
LIN {X 0,Y 601.364,Z 475.147,A -85,B 0,C 180,E1 -813.685,E2 -813.685} C_VEL
LIN {X 0,Y 601.366,Z 469.986,A -85,B 0,C 180,E1 -814.692,E2 -814.692} C_VEL
LIN {X 0,Y 601.383,Z 464.431,A -85,B 0,C 180,E1 -815.532,E2 -815.532} C_VEL
LIN {X 0,Y 601.393,Z 457.152,A -85,B 0,C 180,E1 -816.403,E2 -816.403} C_VEL
LIN {X 0,Y 601.413,Z 449.419,A -85,B 0,C 180,E1 -817.132,E2 -817.132} C_VEL
LIN {X 0,Y 601.424,Z 441.766,A -85,B 0,C 180,E1 -817.723,E2 -817.723} C_VEL
LIN {X 0,Y 601.454,Z 433.727,A -85,B 0,C 180,E1 -818.229,E2 -818.229} C_VEL
LIN {X 0,Y 601.451,Z 425.398,A -85,B 0,C 180,E1 -818.652,E2 -818.652} C_VEL
LIN {X 0,Y 601.446,Z 416.898,A -85,B 0,C 180,E1 -818.991,E2 -818.991} C_VEL
LIN {X 0,Y 601.47,Z 406.766,A -85,B 0,C 180,E1 -819.288,E2 -819.288} C_VEL
LIN {X 0,Y 601.504,Z 395.084,A -85,B 0,C 180,E1 -819.499,E2 -819.499} C_VEL
LIN {X 0,Y 601.454,Z 323.538,A -85,B 0,C 180,E1 -820.349,E2 -820.349} C_VEL
LIN {X 0,Y 601.406,Z 322.757,A -85,B 0,C 180,E1 -820.393,E2 -820.393} C_VEL
LIN {X 0,Y 601.396,Z 304.103,A -85,B 0,C 180,E1 -823.344,E2 -823.344} C_VEL
LIN {X 0,Y 601.482,Z 287.882,A -85,B 0,C 180,E1 -825.937,E2 -825.937} C_VEL
LIN {X 0,Y 601.523,Z 269.923,A -85,B 0,C 180,E1 -828.848,E2 -828.848} C_VEL
LIN {X 0,Y 601.555,Z 256.967,A -85,B 0,C 180,E1 -830.98,E2 -830.98} C_VEL
LIN {X 0,Y 601.387,Z 255.383,A -85,B 0,C 180,E1 -831.284,E2 -831.284} C_VEL
LIN {X 0,Y 601.425,Z 255.379,A -85,B 0,C 180,E1 -834.141,E2 -834.141} C_VEL
LIN {X 0,Y 601.435,Z 255.377,A -85,B 0,C 180,E1 -837.111,E2 -837.111} C_VEL
LIN {X 0,Y 601.393,Z 255.38,A -85,B 0,C 180,E1 -839.394,E2 -839.394} C_VEL
LIN {X 0,Y 601.382,Z 255.38,A -85,B 0,C 180,E1 -841.727,E2 -841.727} C_VEL
LIN {X 0,Y 601.406,Z 255.377,A -85,B 0,C 180,E1 -844.119,E2 -844.119} C_VEL
LIN {X 0,Y 601.431,Z 255.379,A -85,B 0,C 180,E1 -847.381,E2 -847.381} C_VEL
LIN {X 0,Y 601.382,Z 255.38,A -85,B 0,C 180,E1 -849.996,E2 -849.996} C_VEL
LIN {X 0,Y 601.37,Z 255.383,A -85,B 0,C 180,E1 -852.672,E2 -852.672} C_VEL
LIN {X 0,Y 601.388,Z 255.38,A -85,B 0,C 180,E1 -854.532,E2 -854.532} C_VEL
LIN {X 0,Y 601.405,Z 255.389,A -85,B 0,C 180,E1 -857.408,E2 -857.408} C_VEL
LIN {X 0,Y 601.397,Z 255.381,A -85,B 0,C 180,E1 -860.004,E2 -860.004} C_VEL
LIN {X 0,Y 601.417,Z 255.375,A -85,B 0,C 180,E1 -862.618,E2 -862.618} C_VEL
LIN {X 0,Y 601.378,Z 255.382,A -85,B 0,C 180,E1 -865.066,E2 -865.066} C_VEL
LIN {X 0,Y 601.415,Z 255.382,A -85,B 0,C 180,E1 -867.483,E2 -867.483} C_VEL
LIN {X 0,Y 601.438,Z 255.385,A -85,B 0,C 180,E1 -869.847,E2 -869.847} C_VEL
LIN {X 0,Y 601.403,Z 255.376,A -85,B 0,C 180,E1 -872.887,E2 -872.887} C_VEL
LIN {X 0,Y 601.383,Z 255.379,A -85,B 0,C 180,E1 -875.121,E2 -875.121} C_VEL
LIN {X 0,Y 601.4,Z 255.378,A -85,B 0,C 180,E1 -877.394,E2 -877.394} C_VEL
LIN {X 0,Y 601.395,Z 255.389,A -85,B 0,C 180,E1 -880.19,E2 -880.19} C_VEL
LIN {X 0,Y 601.4,Z 255.378,A -85,B 0,C 180,E1 -883.013,E2 -883.013} C_VEL
LIN {X 0,Y 601.394,Z 255.379,A -85,B 0,C 180,E1 -885.794,E2 -885.794} C_VEL
LIN {X 0,Y 601.424,Z 255.386,A -85,B 0,C 180,E1 -888.542,E2 -888.542} C_VEL
LIN {X 0,Y 601.423,Z 255.376,A -85,B 0,C 180,E1 -891.262,E2 -891.262} C_VEL
LIN {X 0,Y 601.439,Z 255.374,A -85,B 0,C 180,E1 -893.324,E2 -893.324} C_VEL
LIN {X 0,Y 601.373,Z 255.381,A -85,B 0,C 180,E1 -895.979,E2 -895.979} C_VEL
LIN {X 0,Y 601.393,Z 255.378,A -85,B 0,C 180,E1 -897.991,E2 -897.991} C_VEL
LIN {X 0,Y 601.415,Z 255.375,A -85,B 0,C 180,E1 -900,E2 -900} C_VEL
LIN {X 0,Y 601.419,Z 255.379,A -85,B 0,C 180,E1 -902.679,E2 -902.679} C_VEL
LIN {X 0,Y 601.431,Z 255.38,A -85,B 0,C 180,E1 -905.364,E2 -905.364} C_VEL
LIN {X 0,Y 601.428,Z 255.374,A -85,B 0,C 180,E1 -908.061,E2 -908.061} C_VEL
LIN {X 0,Y 601.388,Z 255.381,A -85,B 0,C 180,E1 -910.777,E2 -910.777} C_VEL
LIN {X 0,Y 601.395,Z 255.377,A -85,B 0,C 180,E1 -912.36,E2 -912.36} C_VEL
LIN {X 0,Y 600.722,Z 255.466,A -85,B 0,C 180,E1 -912.919,E2 -912.919} C_VEL
LIN {X 0,Y 597.868,Z 255.822,A -85,B 0,C 180,E1 -913.827,E2 -913.827} C_VEL
LIN {X 0,Y 595.464,Z 256.121,A -85,B 0,C 180,E1 -914.557,E2 -914.557} C_VEL
LIN {X 0,Y 594.434,Z 256.25,A -85,B 0,C 180,E1 -915.121,E2 -915.121} C_VEL
LIN {X 0,Y 594.351,Z 256.259,A -85,B 0,C 180,E1 -915.311,E2 -915.311} C_VEL
LIN {X 0,Y 594.366,Z 256.259,A -85,B 0,C 180,E1 -917.905,E2 -917.905} C_VEL
LIN {X 0,Y 594.362,Z 256.255,A -85,B 0,C 180,E1 -920.917,E2 -920.917} C_VEL
LIN {X 0,Y 594.383,Z 256.262,A -85,B 0,C 180,E1 -923.704,E2 -923.704} C_VEL
LIN {X 0,Y 594.37,Z 256.253,A -85,B 0,C 180,E1 -926.7,E2 -926.7} C_VEL
LIN {X 0,Y 594.371,Z 256.253,A -85,B 0,C 180,E1 -928.999,E2 -928.999} C_VEL
LIN {X 0,Y 594.365,Z 256.257,A -85,B 0,C 180,E1 -931.644,E2 -931.644} C_VEL
LIN {X 0,Y 594.391,Z 256.255,A -85,B 0,C 180,E1 -934.579,E2 -934.579} C_VEL
LIN {X 0,Y 594.378,Z 256.253,A -85,B 0,C 180,E1 -937.087,E2 -937.087} C_VEL
LIN {X 0,Y 594.363,Z 256.256,A -85,B 0,C 180,E1 -939.775,E2 -939.775} C_VEL
LIN {X 0,Y 594.363,Z 256.264,A -85,B 0,C 180,E1 -942.376,E2 -942.376} C_VEL
LIN {X 0,Y 594.379,Z 256.457,A -85,B 0,C 180,E1 -943.955,E2 -943.955} C_VEL
LIN {X 0,Y 594.398,Z 268.645,A -85,B 0,C 180,E1 -946.434,E2 -946.434} C_VEL
LIN {X 0,Y 594.338,Z 282.348,A -85,B 0,C 180,E1 -949.183,E2 -949.183} C_VEL
LIN {X 0,Y 594.31,Z 294.353,A -85,B 0,C 180,E1 -951.567,E2 -951.567} C_VEL
LIN {X 0,Y 594.543,Z 303.676,A -85,B 0,C 180,E1 -951.696,E2 -951.696} C_VEL
LIN {X 0,Y 594.52,Z 369.72,A -85,B 0,C 180,E1 -952.507,E2 -952.507} C_VEL
LIN {X 0,Y 594.493,Z 379.111,A -85,B 0,C 180,E1 -952.708,E2 -952.708} C_VEL
LIN {X 0,Y 594.473,Z 388.46,A -85,B 0,C 180,E1 -953.003,E2 -953.003} C_VEL
LIN {X 0,Y 594.45,Z 399.06,A -85,B 0,C 180,E1 -953.459,E2 -953.459} C_VEL
LIN {X 0,Y 594.364,Z 409.514,A -85,B 0,C 180,E1 -954.072,E2 -954.072} C_VEL
LIN {X 0,Y 594.331,Z 417.664,A -85,B 0,C 180,E1 -954.679,E2 -954.679} C_VEL
LIN {X 0,Y 594.336,Z 424.658,A -85,B 0,C 180,E1 -955.315,E2 -955.315} C_VEL
LIN {X 0,Y 594.304,Z 431.348,A -85,B 0,C 180,E1 -956.054,E2 -956.054} C_VEL
LIN {X 0,Y 594.292,Z 438.542,A -85,B 0,C 180,E1 -957.046,E2 -957.046} C_VEL
LIN {X 0,Y 594.264,Z 443.043,A -85,B 0,C 180,E1 -957.848,E2 -957.848} C_VEL
LIN {X 0,Y 594.267,Z 446.582,A -85,B 0,C 180,E1 -958.645,E2 -958.645} C_VEL
LIN {X 0,Y 594.246,Z 449.932,A -85,B 0,C 180,E1 -959.695,E2 -959.695} C_VEL
LIN {X 0,Y 594.229,Z 451.163,A -85,B 0,C 180,E1 -960.217,E2 -960.217} C_VEL
LIN {X 0,Y 594.248,Z 452.457,A -85,B 0,C 180,E1 -961.066,E2 -961.066} C_VEL
LIN {X 0,Y 594.217,Z 452.896,A -85,B 0,C 180,E1 -961.766,E2 -961.766} C_VEL
LIN {X 0,Y 594.259,Z 452.8,A -85,B 0,C 180,E1 -962.534,E2 -962.534} C_VEL
LIN {X 0,Y 594.219,Z 452.084,A -85,B 0,C 180,E1 -963.293,E2 -963.293} C_VEL
LIN {X 0,Y 594.224,Z 450.747,A -85,B 0,C 180,E1 -964.05,E2 -964.05} C_VEL
LIN {X 0,Y 594.25,Z 447.517,A -85,B 0,C 180,E1 -965.176,E2 -965.176} C_VEL
LIN {X 0,Y 594.283,Z 444.379,A -85,B 0,C 180,E1 -965.946,E2 -965.946} C_VEL
LIN {X 0,Y 594.262,Z 439.696,A -85,B 0,C 180,E1 -966.845,E2 -966.845} C_VEL
LIN {X 0,Y 594.294,Z 433.573,A -85,B 0,C 180,E1 -967.765,E2 -967.765} C_VEL
LIN {X 0,Y 594.347,Z 425.746,A -85,B 0,C 180,E1 -968.665,E2 -968.665} C_VEL
LIN {X 0,Y 594.348,Z 418.809,A -85,B 0,C 180,E1 -969.314,E2 -969.314} C_VEL
LIN {X 0,Y 594.362,Z 410.537,A -85,B 0,C 180,E1 -969.946,E2 -969.946} C_VEL
LIN {X 0,Y 594.416,Z 400.118,A -85,B 0,C 180,E1 -970.578,E2 -970.578} C_VEL
LIN {X 0,Y 594.464,Z 389.536,A -85,B 0,C 180,E1 -971.049,E2 -971.049} C_VEL
LIN {X 0,Y 594.48,Z 379.817,A -85,B 0,C 180,E1 -971.364,E2 -971.364} C_VEL
LIN {X 0,Y 594.523,Z 370.738,A -85,B 0,C 180,E1 -971.566,E2 -971.566} C_VEL
LIN {X 0,Y 594.532,Z 333.614,A -85,B 0,C 180,E1 -972.034,E2 -972.034} C_VEL
LIN {X 0,Y 594.412,Z 295.288,A -85,B 0,C 180,E1 -972.497,E2 -972.497} C_VEL
LIN {X 0,Y 594.342,Z 294.265,A -85,B 0,C 180,E1 -972.54,E2 -972.54} C_VEL
LIN {X 0,Y 594.36,Z 278.766,A -85,B 0,C 180,E1 -975.623,E2 -975.623} C_VEL
LIN {X 0,Y 594.399,Z 264.947,A -85,B 0,C 180,E1 -978.405,E2 -978.405} C_VEL
LIN {X 0,Y 594.4,Z 256.253,A -85,B 0,C 180,E1 -980.215,E2 -980.215} C_VEL
LIN {X 0,Y 594.4,Z 256.255,A -85,B 0,C 180,E1 -983.31,E2 -983.31} C_VEL
LIN {X 0,Y 594.353,Z 256.264,A -85,B 0,C 180,E1 -985.932,E2 -985.932} C_VEL
LIN {X 0,Y 594.393,Z 256.259,A -85,B 0,C 180,E1 -987.967,E2 -987.967} C_VEL
LIN {X 0,Y 594.413,Z 256.248,A -85,B 0,C 180,E1 -990.677,E2 -990.677} C_VEL
LIN {X 0,Y 594.384,Z 256.253,A -85,B 0,C 180,E1 -993.389,E2 -993.389} C_VEL
LIN {X 0,Y 594.358,Z 256.266,A -85,B 0,C 180,E1 -996.109,E2 -996.109} C_VEL
LIN {X 0,Y 594.378,Z 256.254,A -85,B 0,C 180,E1 -998.842,E2 -998.842} C_VEL
LIN {X 0,Y 594.387,Z 256.252,A -85,B 0,C 180,E1 -1001.596,E2 -1001.596} C_VEL
LIN {X 0,Y 594.391,Z 256.261,A -85,B 0,C 180,E1 -1004.377,E2 -1004.377} C_VEL
LIN {X 0,Y 594.381,Z 256.253,A -85,B 0,C 180,E1 -1007.193,E2 -1007.193} C_VEL
LIN {X 0,Y 594.372,Z 256.255,A -85,B 0,C 180,E1 -1010.053,E2 -1010.053} C_VEL
LIN {X 0,Y 594.357,Z 256.262,A -85,B 0,C 180,E1 -1012.967,E2 -1012.967} C_VEL
LIN {X 0,Y 594.361,Z 256.259,A -85,B 0,C 180,E1 -1015.193,E2 -1015.193} C_VEL
LIN {X 0,Y 594.384,Z 256.253,A -85,B 0,C 180,E1 -1017.526,E2 -1017.526} C_VEL
LIN {X 0,Y 594.384,Z 256.253,A -85,B 0,C 180,E1 -1020.327,E2 -1020.327} C_VEL
LIN {X 0,Y 594.374,Z 256.262,A -85,B 0,C 180,E1 -1022.949,E2 -1022.949} C_VEL
LIN {X 0,Y 594.345,Z 256.263,A -85,B 0,C 180,E1 -1025.408,E2 -1025.408} C_VEL
LIN {X 0,Y 594.377,Z 256.253,A -85,B 0,C 180,E1 -1027.94,E2 -1027.94} C_VEL
LIN {X 0,Y 594.375,Z 256.255,A -85,B 0,C 180,E1 -1030.821,E2 -1030.821} C_VEL
LIN {X 0,Y 594.36,Z 256.259,A -85,B 0,C 180,E1 -1033.839,E2 -1033.839} C_VEL
LIN {X 0,Y 594.379,Z 256.252,A -85,B 0,C 180,E1 -1036.701,E2 -1036.701} C_VEL
LIN {X 0,Y 594.367,Z 256.26,A -85,B 0,C 180,E1 -1039.433,E2 -1039.433} C_VEL
LIN {X 0,Y 594.382,Z 256.253,A -85,B 0,C 180,E1 -1042.39,E2 -1042.39} C_VEL
LIN {X 0,Y 594.376,Z 256.253,A -85,B 0,C 180,E1 -1044.671,E2 -1044.671} C_VEL
LIN {X 0,Y 594.368,Z 256.253,A -85,B 0,C 180,E1 -1047.087,E2 -1047.087} C_VEL
LIN {X 0,Y 594.388,Z 256.256,A -85,B 0,C 180,E1 -1049.669,E2 -1049.669} C_VEL
LIN {X 0,Y 594.362,Z 256.258,A -85,B 0,C 180,E1 -1052.538,E2 -1052.538} C_VEL
LIN {X 0,Y 594.365,Z 256.256,A -85,B 0,C 180,E1 -1054.806,E2 -1054.806} C_VEL
LIN {X 0,Y 594.353,Z 256.255,A -85,B 0,C 180,E1 -1057.264,E2 -1057.264} C_VEL
LIN {X 0,Y 594.366,Z 256.257,A -85,B 0,C 180,E1 -1059.946,E2 -1059.946} C_VEL
LIN {X 0,Y 594.371,Z 256.259,A -85,B 0,C 180,E1 -1062.806,E2 -1062.806} C_VEL
LIN {X 0,Y 594.375,Z 256.253,A -85,B 0,C 180,E1 -1065.825,E2 -1065.825} C_VEL
LIN {X 0,Y 594.385,Z 256.257,A -85,B 0,C 180,E1 -1068.404,E2 -1068.404} C_VEL
LIN {X 0,Y 594.367,Z 256.258,A -85,B 0,C 180,E1 -1071.158,E2 -1071.158} C_VEL
LIN {X 0,Y 594.382,Z 256.255,A -85,B 0,C 180,E1 -1073.309,E2 -1073.309} C_VEL
LIN {X 0,Y 594.343,Z 256.256,A -85,B 0,C 180,E1 -1075.931,E2 -1075.931} C_VEL
LIN {X 0,Y 594.379,Z 256.256,A -85,B 0,C 180,E1 -1078.645,E2 -1078.645} C_VEL
LIN {X 0,Y 594.367,Z 256.261,A -85,B 0,C 180,E1 -1081.355,E2 -1081.355} C_VEL
LIN {X 0,Y 594.375,Z 256.261,A -85,B 0,C 180,E1 -1083.389,E2 -1083.389} C_VEL
LIN {X 0,Y 594.389,Z 256.26,A -85,B 0,C 180,E1 -1085.428,E2 -1085.428} C_VEL
LIN {X 0,Y 594.366,Z 256.254,A -85,B 0,C 180,E1 -1088.157,E2 -1088.157} C_VEL
LIN {X 0,Y 594.432,Z 256.25,A -85,B 0,C 180,E1 -1091.103,E2 -1091.103} C_VEL
LIN {X 0,Y 594.373,Z 256.253,A -85,B 0,C 180,E1 -1094.377,E2 -1094.377} C_VEL
LIN {X 0,Y 594.368,Z 256.256,A -85,B 0,C 180,E1 -1097.194,E2 -1097.194} C_VEL
LIN {X 0,Y 594.359,Z 256.261,A -85,B 0,C 180,E1 -1100.054,E2 -1100.054} C_VEL
LIN {X 0,Y 594.351,Z 256.255,A -85,B 0,C 180,E1 -1102.968,E2 -1102.968} C_VEL
LIN {X 0,Y 594.365,Z 256.254,A -85,B 0,C 180,E1 -1105.193,E2 -1105.193} C_VEL
LIN {X 0,Y 594.364,Z 256.263,A -85,B 0,C 180,E1 -1108.228,E2 -1108.228} C_VEL
LIN {X 0,Y 594.374,Z 256.257,A -85,B 0,C 180,E1 -1110.56,E2 -1110.56} C_VEL
LIN {X 0,Y 594.365,Z 256.255,A -85,B 0,C 180,E1 -1112.951,E2 -1112.951} C_VEL
LIN {X 0,Y 594.339,Z 256.257,A -85,B 0,C 180,E1 -1115.41,E2 -1115.41} C_VEL
LIN {X 0,Y 594.377,Z 256.255,A -85,B 0,C 180,E1 -1117.941,E2 -1117.941} C_VEL
LIN {X 0,Y 594.365,Z 256.26,A -85,B 0,C 180,E1 -1120.823,E2 -1120.823} C_VEL
LIN {X 0,Y 594.341,Z 256.258,A -85,B 0,C 180,E1 -1123.302,E2 -1123.302} C_VEL
LIN {X 0,Y 594.366,Z 256.256,A -85,B 0,C 180,E1 -1126.161,E2 -1126.161} C_VEL
LIN {X 0,Y 594.367,Z 256.259,A -85,B 0,C 180,E1 -1129.179,E2 -1129.179} C_VEL
LIN {X 0,Y 594.364,Z 256.254,A -85,B 0,C 180,E1 -1132.059,E2 -1132.059} C_VEL
LIN {X 0,Y 594.345,Z 256.261,A -85,B 0,C 180,E1 -1134.677,E2 -1134.677} C_VEL
LIN {X 0,Y 594.369,Z 256.264,A -85,B 0,C 180,E1 -1137.09,E2 -1137.09} C_VEL
LIN {X 0,Y 594.36,Z 256.258,A -85,B 0,C 180,E1 -1139.676,E2 -1139.676} C_VEL
LIN {X 0,Y 594.355,Z 256.258,A -85,B 0,C 180,E1 -1141.773,E2 -1141.773} C_VEL
LIN {X 0,Y 594.334,Z 256.259,A -85,B 0,C 180,E1 -1144.055,E2 -1144.055} C_VEL
LIN {X 0,Y 594.352,Z 256.256,A -85,B 0,C 180,E1 -1146.295,E2 -1146.295} C_VEL
LIN {X 0,Y 594.388,Z 256.371,A -85,B 0,C 180,E1 -1148.655,E2 -1148.655} C_VEL
LIN {X 0,Y 594.566,Z 264.091,A -85,B 0,C 180,E1 -1149.954,E2 -1149.954} C_VEL
LIN {X 0,Y 594.47,Z 281.393,A -85,B 0,C 180,E1 -1152.81,E2 -1152.81} C_VEL
LIN {X 0,Y 594.436,Z 298.696,A -85,B 0,C 180,E1 -1155.625,E2 -1155.625} C_VEL
LIN {X 0,Y 594.341,Z 314.917,A -85,B 0,C 180,E1 -1158.231,E2 -1158.231} C_VEL
LIN {X 0,Y 594.348,Z 322.892,A -85,B 0,C 180,E1 -1159.504,E2 -1159.504} C_VEL
LIN {X 0,Y 594.55,Z 330.691,A -85,B 0,C 180,E1 -1159.615,E2 -1159.615} C_VEL
LIN {X 0,Y 594.522,Z 399.158,A -85,B 0,C 180,E1 -1160.453,E2 -1160.453} C_VEL
LIN {X 0,Y 594.49,Z 408.424,A -85,B 0,C 180,E1 -1160.645,E2 -1160.645} C_VEL
LIN {X 0,Y 594.434,Z 416.898,A -85,B 0,C 180,E1 -1160.902,E2 -1160.902} C_VEL
LIN {X 0,Y 594.422,Z 425.401,A -85,B 0,C 180,E1 -1161.244,E2 -1161.244} C_VEL
LIN {X 0,Y 594.433,Z 433.729,A -85,B 0,C 180,E1 -1161.673,E2 -1161.673} C_VEL
LIN {X 0,Y 594.359,Z 441.767,A -85,B 0,C 180,E1 -1162.185,E2 -1162.185} C_VEL
LIN {X 0,Y 594.354,Z 449.418,A -85,B 0,C 180,E1 -1162.783,E2 -1162.783} C_VEL
LIN {X 0,Y 594.33,Z 457.809,A -85,B 0,C 180,E1 -1163.589,E2 -1163.589} C_VEL
LIN {X 0,Y 594.309,Z 464.433,A -85,B 0,C 180,E1 -1164.401,E2 -1164.401} C_VEL
LIN {X 0,Y 594.276,Z 469.987,A -85,B 0,C 180,E1 -1165.252,E2 -1165.252} C_VEL
LIN {X 0,Y 594.286,Z 475.147,A -85,B 0,C 180,E1 -1166.271,E2 -1166.271} C_VEL
LIN {X 0,Y 594.246,Z 477.788,A -85,B 0,C 180,E1 -1166.949,E2 -1166.949} C_VEL
LIN {X 0,Y 594.241,Z 480.68,A -85,B 0,C 180,E1 -1167.967,E2 -1167.967} C_VEL
LIN {X 0,Y 594.245,Z 481.935,A -85,B 0,C 180,E1 -1168.645,E2 -1168.645} C_VEL
LIN {X 0,Y 594.235,Z 482.712,A -85,B 0,C 180,E1 -1169.322,E2 -1169.322} C_VEL
LIN {X 0,Y 594.233,Z 483,A -85,B 0,C 180,E1 -1170,E2 -1170} C_VEL
LIN {X 0,Y 594.235,Z 482.712,A -85,B 0,C 180,E1 -1170.678,E2 -1170.678} C_VEL
LIN {X 0,Y 594.245,Z 481.935,A -85,B 0,C 180,E1 -1171.355,E2 -1171.355} C_VEL
LIN {X 0,Y 594.241,Z 480.68,A -85,B 0,C 180,E1 -1172.033,E2 -1172.033} C_VEL
LIN {X 0,Y 594.246,Z 477.787,A -85,B 0,C 180,E1 -1173.051,E2 -1173.051} C_VEL
LIN {X 0,Y 594.286,Z 475.147,A -85,B 0,C 180,E1 -1173.729,E2 -1173.729} C_VEL
LIN {X 0,Y 594.276,Z 469.986,A -85,B 0,C 180,E1 -1174.748,E2 -1174.748} C_VEL
LIN {X 0,Y 594.309,Z 464.431,A -85,B 0,C 180,E1 -1175.599,E2 -1175.599} C_VEL
LIN {X 0,Y 594.344,Z 457.151,A -85,B 0,C 180,E1 -1176.479,E2 -1176.479} C_VEL
LIN {X 0,Y 594.354,Z 449.42,A -85,B 0,C 180,E1 -1177.217,E2 -1177.217} C_VEL
LIN {X 0,Y 594.359,Z 441.769,A -85,B 0,C 180,E1 -1177.815,E2 -1177.815} C_VEL
LIN {X 0,Y 594.433,Z 433.73,A -85,B 0,C 180,E1 -1178.327,E2 -1178.327} C_VEL
LIN {X 0,Y 594.422,Z 425.402,A -85,B 0,C 180,E1 -1178.756,E2 -1178.756} C_VEL
LIN {X 0,Y 594.434,Z 416.9,A -85,B 0,C 180,E1 -1179.098,E2 -1179.098} C_VEL
LIN {X 0,Y 594.48,Z 406.766,A -85,B 0,C 180,E1 -1179.398,E2 -1179.398} C_VEL
LIN {X 0,Y 594.522,Z 395.084,A -85,B 0,C 180,E1 -1179.612,E2 -1179.612} C_VEL
LIN {X 0,Y 594.4,Z 323.538,A -85,B 0,C 180,E1 -1180.474,E2 -1180.474} C_VEL
LIN {X 0,Y 594.326,Z 322.757,A -85,B 0,C 180,E1 -1180.518,E2 -1180.518} C_VEL
LIN {X 0,Y 594.364,Z 306.266,A -85,B 0,C 180,E1 -1183.157,E2 -1183.157} C_VEL
LIN {X 0,Y 594.454,Z 290.045,A -85,B 0,C 180,E1 -1185.778,E2 -1185.778} C_VEL
LIN {X 0,Y 594.518,Z 272.742,A -85,B 0,C 180,E1 -1188.612,E2 -1188.612} C_VEL
LIN {X 0,Y 594.517,Z 257.317,A -85,B 0,C 180,E1 -1191.181,E2 -1191.181} C_VEL
LIN {X 0,Y 594.368,Z 256.258,A -85,B 0,C 180,E1 -1191.384,E2 -1191.384} C_VEL
LIN {X 0,Y 594.372,Z 256.263,A -85,B 0,C 180,E1 -1194.43,E2 -1194.43} C_VEL
LIN {X 0,Y 594.354,Z 256.256,A -85,B 0,C 180,E1 -1197.461,E2 -1197.461} C_VEL
LIN {X 0,Y 594.349,Z 256.256,A -85,B 0,C 180,E1 -1199.777,E2 -1199.777} C_VEL
LIN {X 0,Y 594.345,Z 256.257,A -85,B 0,C 180,E1 -1202.147,E2 -1202.147} C_VEL
LIN {X 0,Y 594.369,Z 256.258,A -85,B 0,C 180,E1 -1204.579,E2 -1204.579} C_VEL
LIN {X 0,Y 594.378,Z 256.255,A -85,B 0,C 180,E1 -1207.607,E2 -1207.607} C_VEL
LIN {X 0,Y 594.352,Z 256.258,A -85,B 0,C 180,E1 -1210.567,E2 -1210.567} C_VEL
LIN {X 0,Y 594.363,Z 256.265,A -85,B 0,C 180,E1 -1213.298,E2 -1213.298} C_VEL
LIN {X 0,Y 594.341,Z 256.257,A -85,B 0,C 180,E1 -1216.161,E2 -1216.161} C_VEL
LIN {X 0,Y 594.361,Z 256.254,A -85,B 0,C 180,E1 -1218.535,E2 -1218.535} C_VEL
LIN {X 0,Y 594.368,Z 256.26,A -85,B 0,C 180,E1 -1221.295,E2 -1221.295} C_VEL
LIN {X 0,Y 594.383,Z 256.261,A -85,B 0,C 180,E1 -1223.758,E2 -1223.758} C_VEL
LIN {X 0,Y 594.365,Z 256.256,A -85,B 0,C 180,E1 -1226.238,E2 -1226.238} C_VEL
LIN {X 0,Y 594.355,Z 256.255,A -85,B 0,C 180,E1 -1228.649,E2 -1228.649} C_VEL
LIN {X 0,Y 594.363,Z 256.254,A -85,B 0,C 180,E1 -1231.043,E2 -1231.043} C_VEL
LIN {X 0,Y 594.379,Z 256.263,A -85,B 0,C 180,E1 -1233.975,E2 -1233.975} C_VEL
LIN {X 0,Y 594.37,Z 256.26,A -85,B 0,C 180,E1 -1236.295,E2 -1236.295} C_VEL
LIN {X 0,Y 594.375,Z 256.252,A -85,B 0,C 180,E1 -1239.223,E2 -1239.223} C_VEL
LIN {X 0,Y 594.335,Z 256.265,A -85,B 0,C 180,E1 -1242.094,E2 -1242.094} C_VEL
LIN {X 0,Y 594.355,Z 256.263,A -85,B 0,C 180,E1 -1244.219,E2 -1244.219} C_VEL
LIN {X 0,Y 594.351,Z 256.258,A -85,B 0,C 180,E1 -1247.017,E2 -1247.017} C_VEL
LIN {X 0,Y 594.389,Z 256.253,A -85,B 0,C 180,E1 -1249.095,E2 -1249.095} C_VEL
LIN {X 0,Y 594.365,Z 256.254,A -85,B 0,C 180,E1 -1251.843,E2 -1251.843} C_VEL
LIN {X 0,Y 594.387,Z 256.259,A -85,B 0,C 180,E1 -1254.572,E2 -1254.572} C_VEL
LIN {X 0,Y 594.409,Z 256.251,A -85,B 0,C 180,E1 -1257.289,E2 -1257.289} C_VEL
LIN {X 0,Y 594.385,Z 256.251,A -85,B 0,C 180,E1 -1260,E2 -1260} C_VEL
LIN {X 0,Y 594.387,Z 256.256,A -85,B 0,C 180,E1 -1262.711,E2 -1262.711} C_VEL
LIN {X 0,Y 594.395,Z 256.256,A -85,B 0,C 180,E1 -1265.428,E2 -1265.428} C_VEL
LIN {X 0,Y 594.399,Z 256.249,A -85,B 0,C 180,E1 -1268.157,E2 -1268.157} C_VEL
LIN {X 0,Y 594.365,Z 256.26,A -85,B 0,C 180,E1 -1271.07,E2 -1271.07} C_VEL
LIN {X 0,Y 594.372,Z 256.26,A -85,B 0,C 180,E1 -1273.679,E2 -1273.679} C_VEL
LIN {X 0,Y 594.351,Z 256.259,A -85,B 0,C 180,E1 -1275.311,E2 -1275.311} C_VEL
LIN {X 0,Y 593.687,Z 256.344,A -85,B 0,C 180,E1 -1275.877,E2 -1275.877} C_VEL
LIN {X 0,Y 590.834,Z 256.699,A -85,B 0,C 180,E1 -1276.795,E2 -1276.795} C_VEL
LIN {X 0,Y 588.424,Z 257.005,A -85,B 0,C 180,E1 -1277.534,E2 -1277.534} C_VEL
LIN {X 0,Y 587.391,Z 257.126,A -85,B 0,C 180,E1 -1278.104,E2 -1278.104} C_VEL
LIN {X 0,Y 587.308,Z 257.134,A -85,B 0,C 180,E1 -1278.297,E2 -1278.297} C_VEL
LIN {X 0,Y 587.316,Z 257.133,A -85,B 0,C 180,E1 -1281.038,E2 -1281.038} C_VEL
LIN {X 0,Y 587.311,Z 257.135,A -85,B 0,C 180,E1 -1283.259,E2 -1283.259} C_VEL
LIN {X 0,Y 587.324,Z 257.136,A -85,B 0,C 180,E1 -1285.517,E2 -1285.517} C_VEL
LIN {X 0,Y 587.338,Z 257.138,A -85,B 0,C 180,E1 -1287.818,E2 -1287.818} C_VEL
LIN {X 0,Y 587.334,Z 257.133,A -85,B 0,C 180,E1 -1290.512,E2 -1290.512} C_VEL
LIN {X 0,Y 587.322,Z 257.132,A -85,B 0,C 180,E1 -1293.398,E2 -1293.398} C_VEL
LIN {X 0,Y 587.347,Z 257.133,A -85,B 0,C 180,E1 -1295.896,E2 -1295.896} C_VEL
LIN {X 0,Y 587.325,Z 257.14,A -85,B 0,C 180,E1 -1298.48,E2 -1298.48} C_VEL
LIN {X 0,Y 587.328,Z 257.132,A -85,B 0,C 180,E1 -1301.158,E2 -1301.158} C_VEL
LIN {X 0,Y 587.364,Z 257.225,A -85,B 0,C 180,E1 -1303.891,E2 -1303.891} C_VEL
LIN {X 0,Y 587.346,Z 269.901,A -85,B 0,C 180,E1 -1306.498,E2 -1306.498} C_VEL
LIN {X 0,Y 587.295,Z 282.899,A -85,B 0,C 180,E1 -1309.137,E2 -1309.137} C_VEL
LIN {X 0,Y 587.225,Z 294.379,A -85,B 0,C 180,E1 -1311.445,E2 -1311.445} C_VEL
LIN {X 0,Y 587.557,Z 301.069,A -85,B 0,C 180,E1 -1311.54,E2 -1311.54} C_VEL
LIN {X 0,Y 587.525,Z 369.704,A -85,B 0,C 180,E1 -1312.392,E2 -1312.392} C_VEL
LIN {X 0,Y 587.489,Z 379.029,A -85,B 0,C 180,E1 -1312.594,E2 -1312.594} C_VEL
LIN {X 0,Y 587.471,Z 388.295,A -85,B 0,C 180,E1 -1312.888,E2 -1312.888} C_VEL
LIN {X 0,Y 587.416,Z 398.878,A -85,B 0,C 180,E1 -1313.347,E2 -1313.347} C_VEL
LIN {X 0,Y 587.326,Z 409.823,A -85,B 0,C 180,E1 -1313.998,E2 -1313.998} C_VEL
LIN {X 0,Y 587.279,Z 417.706,A -85,B 0,C 180,E1 -1314.594,E2 -1314.594} C_VEL
LIN {X 0,Y 587.267,Z 423.703,A -85,B 0,C 180,E1 -1315.137,E2 -1315.137} C_VEL
LIN {X 0,Y 587.23,Z 429.625,A -85,B 0,C 180,E1 -1315.773,E2 -1315.773} C_VEL
LIN {X 0,Y 587.196,Z 435.915,A -85,B 0,C 180,E1 -1316.596,E2 -1316.596} C_VEL
LIN {X 0,Y 587.175,Z 440.948,A -85,B 0,C 180,E1 -1317.412,E2 -1317.412} C_VEL
LIN {X 0,Y 587.184,Z 444.936,A -85,B 0,C 180,E1 -1318.223,E2 -1318.223} C_VEL
LIN {X 0,Y 587.159,Z 448.011,A -85,B 0,C 180,E1 -1319.024,E2 -1319.024} C_VEL
LIN {X 0,Y 587.16,Z 450.293,A -85,B 0,C 180,E1 -1319.821,E2 -1319.821} C_VEL
LIN {X 0,Y 587.161,Z 452.246,A -85,B 0,C 180,E1 -1320.9,E2 -1320.9} C_VEL
LIN {X 0,Y 587.138,Z 452.728,A -85,B 0,C 180,E1 -1321.394,E2 -1321.394} C_VEL
LIN {X 0,Y 587.151,Z 452.889,A -85,B 0,C 180,E1 -1322.345,E2 -1322.345} C_VEL
LIN {X 0,Y 587.127,Z 452.571,A -85,B 0,C 180,E1 -1322.945,E2 -1322.945} C_VEL
LIN {X 0,Y 587.116,Z 451.227,A -85,B 0,C 180,E1 -1323.868,E2 -1323.868} C_VEL
LIN {X 0,Y 587.147,Z 448.715,A -85,B 0,C 180,E1 -1324.855,E2 -1324.855} C_VEL
LIN {X 0,Y 587.156,Z 445.576,A -85,B 0,C 180,E1 -1325.722,E2 -1325.722} C_VEL
LIN {X 0,Y 587.185,Z 441.664,A -85,B 0,C 180,E1 -1326.55,E2 -1326.55} C_VEL
LIN {X 0,Y 587.208,Z 437.093,A -85,B 0,C 180,E1 -1327.322,E2 -1327.322} C_VEL
LIN {X 0,Y 587.217,Z 431.933,A -85,B 0,C 180,E1 -1328.038,E2 -1328.038} C_VEL
LIN {X 0,Y 587.272,Z 425.432,A -85,B 0,C 180,E1 -1328.777,E2 -1328.777} C_VEL
LIN {X 0,Y 587.298,Z 418.588,A -85,B 0,C 180,E1 -1329.42,E2 -1329.42} C_VEL
LIN {X 0,Y 587.347,Z 410.252,A -85,B 0,C 180,E1 -1330.062,E2 -1330.062} C_VEL
LIN {X 0,Y 587.391,Z 400.614,A -85,B 0,C 180,E1 -1330.653,E2 -1330.653} C_VEL
LIN {X 0,Y 587.456,Z 389.586,A -85,B 0,C 180,E1 -1331.155,E2 -1331.155} C_VEL
LIN {X 0,Y 587.471,Z 379.957,A -85,B 0,C 180,E1 -1331.472,E2 -1331.472} C_VEL
LIN {X 0,Y 587.52,Z 370.954,A -85,B 0,C 180,E1 -1331.677,E2 -1331.677} C_VEL
LIN {X 0,Y 587.561,Z 337.523,A -85,B 0,C 180,E1 -1332.107,E2 -1332.107} C_VEL
LIN {X 0,Y 587.407,Z 295.486,A -85,B 0,C 180,E1 -1332.621,E2 -1332.621} C_VEL
LIN {X 0,Y 587.277,Z 294.392,A -85,B 0,C 180,E1 -1332.642,E2 -1332.642} C_VEL
LIN {X 0,Y 587.32,Z 278.918,A -85,B 0,C 180,E1 -1335.758,E2 -1335.758} C_VEL
LIN {X 0,Y 587.362,Z 264.91,A -85,B 0,C 180,E1 -1338.614,E2 -1338.614} C_VEL
LIN {X 0,Y 587.365,Z 257.13,A -85,B 0,C 180,E1 -1340.227,E2 -1340.227} C_VEL
LIN {X 0,Y 587.374,Z 257.129,A -85,B 0,C 180,E1 -1343.269,E2 -1343.269} C_VEL
LIN {X 0,Y 587.309,Z 257.142,A -85,B 0,C 180,E1 -1345.883,E2 -1345.883} C_VEL
LIN {X 0,Y 587.364,Z 257.135,A -85,B 0,C 180,E1 -1347.943,E2 -1347.943} C_VEL
LIN {X 0,Y 587.385,Z 257.124,A -85,B 0,C 180,E1 -1350.686,E2 -1350.686} C_VEL
LIN {X 0,Y 587.336,Z 257.131,A -85,B 0,C 180,E1 -1353.43,E2 -1353.43} C_VEL
LIN {X 0,Y 587.359,Z 257.128,A -85,B 0,C 180,E1 -1355.493,E2 -1355.493} C_VEL
LIN {X 0,Y 587.364,Z 257.137,A -85,B 0,C 180,E1 -1358.255,E2 -1358.255} C_VEL
LIN {X 0,Y 587.35,Z 257.128,A -85,B 0,C 180,E1 -1361.133,E2 -1361.133} C_VEL
LIN {X 0,Y 587.366,Z 257.134,A -85,B 0,C 180,E1 -1364.26,E2 -1364.26} C_VEL
LIN {X 0,Y 587.345,Z 257.128,A -85,B 0,C 180,E1 -1367.406,E2 -1367.406} C_VEL
LIN {X 0,Y 587.312,Z 257.132,A -85,B 0,C 180,E1 -1369.575,E2 -1369.575} C_VEL
LIN {X 0,Y 587.338,Z 257.137,A -85,B 0,C 180,E1 -1372.513,E2 -1372.513} C_VEL
LIN {X 0,Y 587.346,Z 257.139,A -85,B 0,C 180,E1 -1374.758,E2 -1374.758} C_VEL
LIN {X 0,Y 587.345,Z 257.128,A -85,B 0,C 180,E1 -1377.817,E2 -1377.817} C_VEL
LIN {X 0,Y 587.335,Z 257.133,A -85,B 0,C 180,E1 -1380.509,E2 -1380.509} C_VEL
LIN {X 0,Y 587.324,Z 257.137,A -85,B 0,C 180,E1 -1383.396,E2 -1383.396} C_VEL
LIN {X 0,Y 587.286,Z 257.136,A -85,B 0,C 180,E1 -1385.899,E2 -1385.899} C_VEL
LIN {X 0,Y 587.322,Z 257.131,A -85,B 0,C 180,E1 -1388.479,E2 -1388.479} C_VEL
LIN {X 0,Y 587.332,Z 257.137,A -85,B 0,C 180,E1 -1391.156,E2 -1391.156} C_VEL
LIN {X 0,Y 587.319,Z 257.133,A -85,B 0,C 180,E1 -1394.112,E2 -1394.112} C_VEL
LIN {X 0,Y 587.33,Z 257.132,A -85,B 0,C 180,E1 -1396.995,E2 -1396.995} C_VEL
LIN {X 0,Y 587.313,Z 257.138,A -85,B 0,C 180,E1 -1399.98,E2 -1399.98} C_VEL
LIN {X 0,Y 587.337,Z 257.131,A -85,B 0,C 180,E1 -1402.392,E2 -1402.392} C_VEL
LIN {X 0,Y 587.342,Z 257.129,A -85,B 0,C 180,E1 -1404.945,E2 -1404.945} C_VEL
LIN {X 0,Y 587.329,Z 257.133,A -85,B 0,C 180,E1 -1407.42,E2 -1407.42} C_VEL
LIN {X 0,Y 587.335,Z 257.137,A -85,B 0,C 180,E1 -1409.83,E2 -1409.83} C_VEL
LIN {X 0,Y 587.34,Z 257.137,A -85,B 0,C 180,E1 -1412.306,E2 -1412.306} C_VEL
LIN {X 0,Y 587.328,Z 257.136,A -85,B 0,C 180,E1 -1414.483,E2 -1414.483} C_VEL
LIN {X 0,Y 587.307,Z 257.133,A -85,B 0,C 180,E1 -1417.13,E2 -1417.13} C_VEL
LIN {X 0,Y 587.319,Z 257.133,A -85,B 0,C 180,E1 -1419.695,E2 -1419.695} C_VEL
LIN {X 0,Y 587.342,Z 257.138,A -85,B 0,C 180,E1 -1422.594,E2 -1422.594} C_VEL
LIN {X 0,Y 587.351,Z 257.128,A -85,B 0,C 180,E1 -1425.739,E2 -1425.739} C_VEL
LIN {X 0,Y 587.333,Z 257.138,A -85,B 0,C 180,E1 -1428.866,E2 -1428.866} C_VEL
LIN {X 0,Y 587.352,Z 257.127,A -85,B 0,C 180,E1 -1431.744,E2 -1431.744} C_VEL
LIN {X 0,Y 587.359,Z 257.131,A -85,B 0,C 180,E1 -1434.507,E2 -1434.507} C_VEL
LIN {X 0,Y 587.357,Z 257.133,A -85,B 0,C 180,E1 -1437.257,E2 -1437.257} C_VEL
LIN {X 0,Y 587.357,Z 257.127,A -85,B 0,C 180,E1 -1440,E2 -1440} C_VEL
LIN {X 0,Y 587.374,Z 257.128,A -85,B 0,C 180,E1 -1442.743,E2 -1442.743} C_VEL
LIN {X 0,Y 587.351,Z 257.135,A -85,B 0,C 180,E1 -1445.493,E2 -1445.493} C_VEL
LIN {X 0,Y 587.329,Z 257.13,A -85,B 0,C 180,E1 -1448.256,E2 -1448.256} C_VEL
LIN {X 0,Y 587.379,Z 257.129,A -85,B 0,C 180,E1 -1451.157,E2 -1451.157} C_VEL
LIN {X 0,Y 587.349,Z 257.129,A -85,B 0,C 180,E1 -1454.261,E2 -1454.261} C_VEL
LIN {X 0,Y 587.339,Z 257.134,A -85,B 0,C 180,E1 -1457.406,E2 -1457.406} C_VEL
LIN {X 0,Y 587.309,Z 257.136,A -85,B 0,C 180,E1 -1460.305,E2 -1460.305} C_VEL
LIN {X 0,Y 587.311,Z 257.134,A -85,B 0,C 180,E1 -1463.259,E2 -1463.259} C_VEL
LIN {X 0,Y 587.326,Z 257.134,A -85,B 0,C 180,E1 -1465.517,E2 -1465.517} C_VEL
LIN {X 0,Y 587.334,Z 257.136,A -85,B 0,C 180,E1 -1467.818,E2 -1467.818} C_VEL
LIN {X 0,Y 587.331,Z 257.135,A -85,B 0,C 180,E1 -1470.512,E2 -1470.512} C_VEL
LIN {X 0,Y 587.322,Z 257.131,A -85,B 0,C 180,E1 -1473.397,E2 -1473.397} C_VEL
LIN {X 0,Y 587.305,Z 257.136,A -85,B 0,C 180,E1 -1475.899,E2 -1475.899} C_VEL
LIN {X 0,Y 587.317,Z 257.143,A -85,B 0,C 180,E1 -1478.48,E2 -1478.48} C_VEL
LIN {X 0,Y 587.322,Z 257.133,A -85,B 0,C 180,E1 -1481.158,E2 -1481.158} C_VEL
LIN {X 0,Y 587.308,Z 257.135,A -85,B 0,C 180,E1 -1484.113,E2 -1484.113} C_VEL
LIN {X 0,Y 587.295,Z 257.142,A -85,B 0,C 180,E1 -1486.993,E2 -1486.993} C_VEL
LIN {X 0,Y 587.302,Z 257.134,A -85,B 0,C 180,E1 -1489.746,E2 -1489.746} C_VEL
LIN {X 0,Y 587.334,Z 257.132,A -85,B 0,C 180,E1 -1492.393,E2 -1492.393} C_VEL
LIN {X 0,Y 587.332,Z 257.132,A -85,B 0,C 180,E1 -1495.655,E2 -1495.655} C_VEL
LIN {X 0,Y 587.326,Z 257.131,A -85,B 0,C 180,E1 -1498.231,E2 -1498.231} C_VEL
LIN {X 0,Y 587.341,Z 257.133,A -85,B 0,C 180,E1 -1500.868,E2 -1500.868} C_VEL
LIN {X 0,Y 587.3,Z 257.138,A -85,B 0,C 180,E1 -1503.831,E2 -1503.831} C_VEL
LIN {X 0,Y 587.301,Z 257.135,A -85,B 0,C 180,E1 -1506.741,E2 -1506.741} C_VEL
LIN {X 0,Y 587.356,Z 257.334,A -85,B 0,C 180,E1 -1508.551,E2 -1508.551} C_VEL
LIN {X 0,Y 587.6,Z 263.009,A -85,B 0,C 180,E1 -1509.523,E2 -1509.523} C_VEL
LIN {X 0,Y 587.48,Z 279.23,A -85,B 0,C 180,E1 -1512.239,E2 -1512.239} C_VEL
LIN {X 0,Y 587.419,Z 295.451,A -85,B 0,C 180,E1 -1514.917,E2 -1514.917} C_VEL
LIN {X 0,Y 587.319,Z 314.917,A -85,B 0,C 180,E1 -1518.088,E2 -1518.088} C_VEL
LIN {X 0,Y 587.273,Z 322.892,A -85,B 0,C 180,E1 -1519.376,E2 -1519.376} C_VEL
LIN {X 0,Y 587.588,Z 328.902,A -85,B 0,C 180,E1 -1519.469,E2 -1519.469} C_VEL
LIN {X 0,Y 587.531,Z 399.156,A -85,B 0,C 180,E1 -1520.338,E2 -1520.338} C_VEL
LIN {X 0,Y 587.47,Z 408.424,A -85,B 0,C 180,E1 -1520.532,E2 -1520.532} C_VEL
LIN {X 0,Y 587.438,Z 416.9,A -85,B 0,C 180,E1 -1520.792,E2 -1520.792} C_VEL
LIN {X 0,Y 587.396,Z 425.404,A -85,B 0,C 180,E1 -1521.139,E2 -1521.139} C_VEL
LIN {X 0,Y 587.402,Z 433.732,A -85,B 0,C 180,E1 -1521.572,E2 -1521.572} C_VEL
LIN {X 0,Y 587.33,Z 441.769,A -85,B 0,C 180,E1 -1522.091,E2 -1522.091} C_VEL
LIN {X 0,Y 587.288,Z 449.419,A -85,B 0,C 180,E1 -1522.695,E2 -1522.695} C_VEL
LIN {X 0,Y 587.281,Z 457.809,A -85,B 0,C 180,E1 -1523.512,E2 -1523.512} C_VEL
LIN {X 0,Y 587.238,Z 464.434,A -85,B 0,C 180,E1 -1524.334,E2 -1524.334} C_VEL
LIN {X 0,Y 587.185,Z 469.987,A -85,B 0,C 180,E1 -1525.194,E2 -1525.194} C_VEL
LIN {X 0,Y 587.21,Z 475.148,A -85,B 0,C 180,E1 -1526.226,E2 -1526.226} C_VEL
LIN {X 0,Y 587.155,Z 477.788,A -85,B 0,C 180,E1 -1526.912,E2 -1526.912} C_VEL
LIN {X 0,Y 587.141,Z 480.68,A -85,B 0,C 180,E1 -1527.942,E2 -1527.942} C_VEL
LIN {X 0,Y 587.145,Z 481.936,A -85,B 0,C 180,E1 -1528.628,E2 -1528.628} C_VEL
LIN {X 0,Y 587.136,Z 482.712,A -85,B 0,C 180,E1 -1529.314,E2 -1529.314} C_VEL
LIN {X 0,Y 587.134,Z 483,A -85,B 0,C 180,E1 -1530,E2 -1530} C_VEL
LIN {X 0,Y 587.136,Z 482.711,A -85,B 0,C 180,E1 -1530.686,E2 -1530.686} C_VEL
LIN {X 0,Y 587.145,Z 481.936,A -85,B 0,C 180,E1 -1531.372,E2 -1531.372} C_VEL
LIN {X 0,Y 587.14,Z 480.68,A -85,B 0,C 180,E1 -1532.058,E2 -1532.058} C_VEL
LIN {X 0,Y 587.155,Z 477.788,A -85,B 0,C 180,E1 -1533.088,E2 -1533.088} C_VEL
LIN {X 0,Y 587.21,Z 475.148,A -85,B 0,C 180,E1 -1533.774,E2 -1533.774} C_VEL
LIN {X 0,Y 587.185,Z 469.986,A -85,B 0,C 180,E1 -1534.806,E2 -1534.806} C_VEL
LIN {X 0,Y 587.238,Z 464.432,A -85,B 0,C 180,E1 -1535.666,E2 -1535.666} C_VEL
LIN {X 0,Y 587.269,Z 456.287,A -85,B 0,C 180,E1 -1536.645,E2 -1536.645} C_VEL
LIN {X 0,Y 587.292,Z 448.408,A -85,B 0,C 180,E1 -1537.391,E2 -1537.391} C_VEL
LIN {X 0,Y 587.343,Z 440.553,A -85,B 0,C 180,E1 -1537.996,E2 -1537.996} C_VEL
LIN {X 0,Y 587.439,Z 430.739,A -85,B 0,C 180,E1 -1538.6,E2 -1538.6} C_VEL
LIN {X 0,Y 587.439,Z 419.308,A -85,B 0,C 180,E1 -1539.121,E2 -1539.121} C_VEL
LIN {X 0,Y 587.469,Z 409.257,A -85,B 0,C 180,E1 -1539.446,E2 -1539.446} C_VEL
LIN {X 0,Y 587.526,Z 400.463,A -85,B 0,C 180,E1 -1539.64,E2 -1539.64} C_VEL
LIN {X 0,Y 587.582,Z 332.481,A -85,B 0,C 180,E1 -1540.488,E2 -1540.488} C_VEL
LIN {X 0,Y 587.325,Z 323.538,A -85,B 0,C 180,E1 -1540.601,E2 -1540.601} C_VEL
LIN {X 0,Y 587.264,Z 322.757,A -85,B 0,C 180,E1 -1540.646,E2 -1540.646} C_VEL
LIN {X 0,Y 587.333,Z 306.266,A -85,B 0,C 180,E1 -1543.317,E2 -1543.317} C_VEL
LIN {X 0,Y 587.454,Z 288.963,A -85,B 0,C 180,E1 -1546.149,E2 -1546.149} C_VEL
LIN {X 0,Y 587.544,Z 271.222,A -85,B 0,C 180,E1 -1549.096,E2 -1549.096} C_VEL
LIN {X 0,Y 587.584,Z 259.329,A -85,B 0,C 180,E1 -1551.101,E2 -1551.101} C_VEL
LIN {X 0,Y 587.321,Z 257.137,A -85,B 0,C 180,E1 -1551.497,E2 -1551.497} C_VEL
LIN {X 0,Y 587.304,Z 257.137,A -85,B 0,C 180,E1 -1554.007,E2 -1554.007} C_VEL
LIN {X 0,Y 587.3,Z 257.139,A -85,B 0,C 180,E1 -1556.28,E2 -1556.28} C_VEL
LIN {X 0,Y 587.34,Z 257.134,A -85,B 0,C 180,E1 -1559.132,E2 -1559.132} C_VEL
LIN {X 0,Y 587.334,Z 257.13,A -85,B 0,C 180,E1 -1561.834,E2 -1561.834} C_VEL
LIN {X 0,Y 587.331,Z 257.132,A -85,B 0,C 180,E1 -1564.345,E2 -1564.345} C_VEL
LIN {X 0,Y 587.334,Z 257.133,A -85,B 0,C 180,E1 -1567.607,E2 -1567.607} C_VEL
LIN {X 0,Y 587.302,Z 257.134,A -85,B 0,C 180,E1 -1570.254,E2 -1570.254} C_VEL
LIN {X 0,Y 587.302,Z 257.143,A -85,B 0,C 180,E1 -1573.117,E2 -1573.117} C_VEL
LIN {X 0,Y 587.299,Z 257.135,A -85,B 0,C 180,E1 -1576.047,E2 -1576.047} C_VEL
LIN {X 0,Y 587.324,Z 257.133,A -85,B 0,C 180,E1 -1578.924,E2 -1578.924} C_VEL
LIN {X 0,Y 587.316,Z 257.143,A -85,B 0,C 180,E1 -1581.52,E2 -1581.52} C_VEL
LIN {X 0,Y 587.305,Z 257.137,A -85,B 0,C 180,E1 -1584.101,E2 -1584.101} C_VEL
LIN {X 0,Y 587.325,Z 257.13,A -85,B 0,C 180,E1 -1586.888,E2 -1586.888} C_VEL
LIN {X 0,Y 587.332,Z 257.141,A -85,B 0,C 180,E1 -1589.83,E2 -1589.83} C_VEL
LIN {X 0,Y 587.338,Z 257.133,A -85,B 0,C 180,E1 -1592.306,E2 -1592.306} C_VEL
LIN {X 0,Y 587.325,Z 257.134,A -85,B 0,C 180,E1 -1594.483,E2 -1594.483} C_VEL
LIN {X 0,Y 587.323,Z 257.132,A -85,B 0,C 180,E1 -1597.486,E2 -1597.486} C_VEL
LIN {X 0,Y 587.328,Z 257.138,A -85,B 0,C 180,E1 -1600.425,E2 -1600.425} C_VEL
LIN {X 0,Y 587.307,Z 257.132,A -85,B 0,C 180,E1 -1603.31,E2 -1603.31} C_VEL
LIN {X 0,Y 587.338,Z 257.135,A -85,B 0,C 180,E1 -1606.154,E2 -1606.154} C_VEL
LIN {X 0,Y 587.378,Z 257.127,A -85,B 0,C 180,E1 -1608.963,E2 -1608.963} C_VEL
LIN {X 0,Y 587.328,Z 257.13,A -85,B 0,C 180,E1 -1611.744,E2 -1611.744} C_VEL
LIN {X 0,Y 587.349,Z 257.135,A -85,B 0,C 180,E1 -1614.507,E2 -1614.507} C_VEL
LIN {X 0,Y 587.373,Z 257.128,A -85,B 0,C 180,E1 -1617.257,E2 -1617.257} C_VEL
LIN {X 0,Y 587.355,Z 257.127,A -85,B 0,C 180,E1 -1620,E2 -1620} C_VEL
LIN {X 0,Y 587.354,Z 257.132,A -85,B 0,C 180,E1 -1622.743,E2 -1622.743} C_VEL
LIN {X 0,Y 587.358,Z 257.131,A -85,B 0,C 180,E1 -1625.493,E2 -1625.493} C_VEL
LIN {X 0,Y 587.351,Z 257.127,A -85,B 0,C 180,E1 -1628.256,E2 -1628.256} C_VEL
LIN {X 0,Y 587.332,Z 257.137,A -85,B 0,C 180,E1 -1631.134,E2 -1631.134} C_VEL
LIN {X 0,Y 587.351,Z 257.128,A -85,B 0,C 180,E1 -1634.261,E2 -1634.261} C_VEL
LIN {X 0,Y 587.337,Z 257.137,A -85,B 0,C 180,E1 -1637.406,E2 -1637.406} C_VEL
LIN {X 0,Y 587.308,Z 257.134,A -85,B 0,C 180,E1 -1638.297,E2 -1638.297} C_VEL
LIN {X 0,Y 586.652,Z 257.216,A -85,B 0,C 180,E1 -1638.869,E2 -1638.869} C_VEL
LIN {X 0,Y 583.823,Z 257.576,A -85,B 0,C 180,E1 -1639.797,E2 -1639.797} C_VEL
LIN {X 0,Y 581.416,Z 257.875,A -85,B 0,C 180,E1 -1640.544,E2 -1640.544} C_VEL
LIN {X 0,Y 580.365,Z 258.003,A -85,B 0,C 180,E1 -1641.12,E2 -1641.12} C_VEL
LIN {X 0,Y 580.27,Z 258.014,A -85,B 0,C 180,E1 -1641.316,E2 -1641.316} C_VEL
LIN {X 0,Y 580.269,Z 258.017,A -85,B 0,C 180,E1 -1643.559,E2 -1643.559} C_VEL
LIN {X 0,Y 580.315,Z 258.008,A -85,B 0,C 180,E1 -1646.342,E2 -1646.342} C_VEL
LIN {X 0,Y 580.294,Z 258.008,A -85,B 0,C 180,E1 -1649.311,E2 -1649.311} C_VEL
LIN {X 0,Y 580.288,Z 258.017,A -85,B 0,C 180,E1 -1652.201,E2 -1652.201} C_VEL
LIN {X 0,Y 580.293,Z 258.01,A -85,B 0,C 180,E1 -1654.696,E2 -1654.696} C_VEL
LIN {X 0,Y 580.291,Z 258.007,A -85,B 0,C 180,E1 -1657.269,E2 -1657.269} C_VEL
LIN {X 0,Y 580.289,Z 258.017,A -85,B 0,C 180,E1 -1660.272,E2 -1660.272} C_VEL
LIN {X 0,Y 580.272,Z 258.017,A -85,B 0,C 180,E1 -1662.707,E2 -1662.707} C_VEL
LIN {X 0,Y 580.322,Z 258.041,A -85,B 0,C 180,E1 -1663.834,E2 -1663.834} C_VEL
LIN {X 0,Y 580.32,Z 270.108,A -85,B 0,C 180,E1 -1666.348,E2 -1666.348} C_VEL
LIN {X 0,Y 580.226,Z 283.754,A -85,B 0,C 180,E1 -1669.152,E2 -1669.152} C_VEL
LIN {X 0,Y 580.185,Z 294.457,A -85,B 0,C 180,E1 -1671.323,E2 -1671.323} C_VEL
LIN {X 0,Y 580.587,Z 300.515,A -85,B 0,C 180,E1 -1671.405,E2 -1671.405} C_VEL
LIN {X 0,Y 580.534,Z 370.39,A -85,B 0,C 180,E1 -1672.286,E2 -1672.286} C_VEL
LIN {X 0,Y 580.502,Z 380.451,A -85,B 0,C 180,E1 -1672.516,E2 -1672.516} C_VEL
LIN {X 0,Y 580.43,Z 392.263,A -85,B 0,C 180,E1 -1672.929,E2 -1672.929} C_VEL
LIN {X 0,Y 580.389,Z 401.992,A -85,B 0,C 180,E1 -1673.413,E2 -1673.413} C_VEL
LIN {X 0,Y 580.271,Z 410.527,A -85,B 0,C 180,E1 -1673.95,E2 -1673.95} C_VEL
LIN {X 0,Y 580.228,Z 418.355,A -85,B 0,C 180,E1 -1674.559,E2 -1674.559} C_VEL
LIN {X 0,Y 580.226,Z 425.085,A -85,B 0,C 180,E1 -1675.195,E2 -1675.195} C_VEL
LIN {X 0,Y 580.146,Z 431.499,A -85,B 0,C 180,E1 -1675.926,E2 -1675.926} C_VEL
LIN {X 0,Y 580.106,Z 437.161,A -85,B 0,C 180,E1 -1676.714,E2 -1676.714} C_VEL
LIN {X 0,Y 580.096,Z 443.243,A -85,B 0,C 180,E1 -1677.788,E2 -1677.788} C_VEL
LIN {X 0,Y 580.073,Z 446.735,A -85,B 0,C 180,E1 -1678.603,E2 -1678.603} C_VEL
LIN {X 0,Y 580.087,Z 449.387,A -85,B 0,C 180,E1 -1679.414,E2 -1679.414} C_VEL
LIN {X 0,Y 580.048,Z 451.259,A -85,B 0,C 180,E1 -1680.215,E2 -1680.215} C_VEL
LIN {X 0,Y 580.052,Z 452.417,A -85,B 0,C 180,E1 -1681.012,E2 -1681.012} C_VEL
LIN {X 0,Y 580.042,Z 452.96,A -85,B 0,C 180,E1 -1682.19,E2 -1682.19} C_VEL
LIN {X 0,Y 580.042,Z 451.543,A -85,B 0,C 180,E1 -1683.716,E2 -1683.716} C_VEL
LIN {X 0,Y 580.053,Z 448.649,A -85,B 0,C 180,E1 -1684.909,E2 -1684.909} C_VEL
LIN {X 0,Y 580.062,Z 445.984,A -85,B 0,C 180,E1 -1685.674,E2 -1685.674} C_VEL
LIN {X 0,Y 580.102,Z 442.59,A -85,B 0,C 180,E1 -1686.435,E2 -1686.435} C_VEL
LIN {X 0,Y 580.142,Z 437.135,A -85,B 0,C 180,E1 -1687.38,E2 -1687.38} C_VEL
LIN {X 0,Y 580.153,Z 431.773,A -85,B 0,C 180,E1 -1688.13,E2 -1688.13} C_VEL
LIN {X 0,Y 580.208,Z 424.68,A -85,B 0,C 180,E1 -1688.937,E2 -1688.937} C_VEL
LIN {X 0,Y 580.233,Z 417.296,A -85,B 0,C 180,E1 -1689.622,E2 -1689.622} C_VEL
LIN {X 0,Y 580.322,Z 407.32,A -85,B 0,C 180,E1 -1690.363,E2 -1690.363} C_VEL
LIN {X 0,Y 580.385,Z 397.46,A -85,B 0,C 180,E1 -1690.917,E2 -1690.917} C_VEL
LIN {X 0,Y 580.449,Z 387.801,A -85,B 0,C 180,E1 -1691.332,E2 -1691.332} C_VEL
LIN {X 0,Y 580.47,Z 378.361,A -85,B 0,C 180,E1 -1691.629,E2 -1691.629} C_VEL
LIN {X 0,Y 580.53,Z 368.443,A -85,B 0,C 180,E1 -1691.837,E2 -1691.837} C_VEL
LIN {X 0,Y 580.573,Z 297.108,A -85,B 0,C 180,E1 -1692.727,E2 -1692.727} C_VEL
LIN {X 0,Y 580.206,Z 294.335,A -85,B 0,C 180,E1 -1692.784,E2 -1692.784} C_VEL
LIN {X 0,Y 580.244,Z 280.079,A -85,B 0,C 180,E1 -1695.69,E2 -1695.69} C_VEL
LIN {X 0,Y 580.316,Z 266.579,A -85,B 0,C 180,E1 -1698.474,E2 -1698.474} C_VEL
LIN {X 0,Y 580.314,Z 258.008,A -85,B 0,C 180,E1 -1700.283,E2 -1700.283} C_VEL
LIN {X 0,Y 580.349,Z 258.004,A -85,B 0,C 180,E1 -1703.226,E2 -1703.226} C_VEL
LIN {X 0,Y 580.265,Z 258.02,A -85,B 0,C 180,E1 -1705.833,E2 -1705.833} C_VEL
LIN {X 0,Y 580.336,Z 258.011,A -85,B 0,C 180,E1 -1707.918,E2 -1707.918} C_VEL
LIN {X 0,Y 580.357,Z 257.999,A -85,B 0,C 180,E1 -1710.694,E2 -1710.694} C_VEL
LIN {X 0,Y 580.287,Z 258.01,A -85,B 0,C 180,E1 -1713.472,E2 -1713.472} C_VEL
LIN {X 0,Y 580.324,Z 258.005,A -85,B 0,C 180,E1 -1715.56,E2 -1715.56} C_VEL
LIN {X 0,Y 580.327,Z 258.011,A -85,B 0,C 180,E1 -1718.356,E2 -1718.356} C_VEL
LIN {X 0,Y 580.302,Z 258.006,A -85,B 0,C 180,E1 -1721.191,E2 -1721.191} C_VEL
LIN {X 0,Y 580.326,Z 258.007,A -85,B 0,C 180,E1 -1724.017,E2 -1724.017} C_VEL
LIN {X 0,Y 580.314,Z 258.008,A -85,B 0,C 180,E1 -1726.913,E2 -1726.913} C_VEL
LIN {X 0,Y 580.287,Z 258.008,A -85,B 0,C 180,E1 -1729.822,E2 -1729.822} C_VEL
LIN {X 0,Y 580.27,Z 258.011,A -85,B 0,C 180,E1 -1732.052,E2 -1732.052} C_VEL
LIN {X 0,Y 580.3,Z 258.012,A -85,B 0,C 180,E1 -1735.079,E2 -1735.079} C_VEL
LIN {X 0,Y 580.297,Z 258.007,A -85,B 0,C 180,E1 -1738.185,E2 -1738.185} C_VEL
LIN {X 0,Y 580.282,Z 258.014,A -85,B 0,C 180,E1 -1740.694,E2 -1740.694} C_VEL
LIN {X 0,Y 580.28,Z 258.015,A -85,B 0,C 180,E1 -1743.312,E2 -1743.312} C_VEL
LIN {X 0,Y 580.241,Z 258.015,A -85,B 0,C 180,E1 -1745.755,E2 -1745.755} C_VEL
LIN {X 0,Y 580.282,Z 258.008,A -85,B 0,C 180,E1 -1748.145,E2 -1748.145} C_VEL
LIN {X 0,Y 580.293,Z 258.009,A -85,B 0,C 180,E1 -1750.842,E2 -1750.842} C_VEL
LIN {X 0,Y 580.272,Z 258.017,A -85,B 0,C 180,E1 -1753.657,E2 -1753.657} C_VEL
LIN {X 0,Y 580.285,Z 258.008,A -85,B 0,C 180,E1 -1756.607,E2 -1756.607} C_VEL
LIN {X 0,Y 580.293,Z 258.01,A -85,B 0,C 180,E1 -1759.156,E2 -1759.156} C_VEL
LIN {X 0,Y 580.283,Z 258.016,A -85,B 0,C 180,E1 -1761.926,E2 -1761.926} C_VEL
LIN {X 0,Y 580.297,Z 258.008,A -85,B 0,C 180,E1 -1764.456,E2 -1764.456} C_VEL
LIN {X 0,Y 580.28,Z 258.008,A -85,B 0,C 180,E1 -1766.974,E2 -1766.974} C_VEL
LIN {X 0,Y 580.292,Z 258.009,A -85,B 0,C 180,E1 -1769.425,E2 -1769.425} C_VEL
LIN {X 0,Y 580.309,Z 258.016,A -85,B 0,C 180,E1 -1772.136,E2 -1772.136} C_VEL
LIN {X 0,Y 580.297,Z 258.007,A -85,B 0,C 180,E1 -1774.92,E2 -1774.92} C_VEL
LIN {X 0,Y 580.262,Z 258.015,A -85,B 0,C 180,E1 -1777.947,E2 -1777.947} C_VEL
LIN {X 0,Y 580.286,Z 258.011,A -85,B 0,C 180,E1 -1780.913,E2 -1780.913} C_VEL
LIN {X 0,Y 580.272,Z 258.01,A -85,B 0,C 180,E1 -1783.825,E2 -1783.825} C_VEL
LIN {X 0,Y 580.314,Z 258.006,A -85,B 0,C 180,E1 -1785.983,E2 -1785.983} C_VEL
LIN {X 0,Y 580.29,Z 258.016,A -85,B 0,C 180,E1 -1788.827,E2 -1788.827} C_VEL
LIN {X 0,Y 580.315,Z 258.004,A -85,B 0,C 180,E1 -1791.644,E2 -1791.644} C_VEL
LIN {X 0,Y 580.324,Z 258.006,A -85,B 0,C 180,E1 -1794.44,E2 -1794.44} C_VEL
LIN {X 0,Y 580.324,Z 258.01,A -85,B 0,C 180,E1 -1797.223,E2 -1797.223} C_VEL
LIN {X 0,Y 580.327,Z 258.002,A -85,B 0,C 180,E1 -1800,E2 -1800} C_VEL
LIN {X 0,Y 580.338,Z 258.005,A -85,B 0,C 180,E1 -1802.776,E2 -1802.776} C_VEL
LIN {X 0,Y 580.315,Z 258.01,A -85,B 0,C 180,E1 -1805.56,E2 -1805.56} C_VEL
LIN {X 0,Y 580.3,Z 258.006,A -85,B 0,C 180,E1 -1808.356,E2 -1808.356} C_VEL
LIN {X 0,Y 580.326,Z 258.008,A -85,B 0,C 180,E1 -1811.212,E2 -1811.212} C_VEL
LIN {X 0,Y 580.3,Z 258.007,A -85,B 0,C 180,E1 -1814.339,E2 -1814.339} C_VEL
LIN {X 0,Y 580.297,Z 258.007,A -85,B 0,C 180,E1 -1816.914,E2 -1816.914} C_VEL
LIN {X 0,Y 580.289,Z 258.019,A -85,B 0,C 180,E1 -1819.823,E2 -1819.823} C_VEL
LIN {X 0,Y 580.281,Z 258.008,A -85,B 0,C 180,E1 -1822.803,E2 -1822.803} C_VEL
LIN {X 0,Y 580.296,Z 258.006,A -85,B 0,C 180,E1 -1825.08,E2 -1825.08} C_VEL
LIN {X 0,Y 580.285,Z 258.018,A -85,B 0,C 180,E1 -1828.186,E2 -1828.186} C_VEL
LIN {X 0,Y 580.276,Z 258.012,A -85,B 0,C 180,E1 -1830.696,E2 -1830.696} C_VEL
LIN {X 0,Y 580.291,Z 258.007,A -85,B 0,C 180,E1 -1833.317,E2 -1833.317} C_VEL
LIN {X 0,Y 580.262,Z 258.012,A -85,B 0,C 180,E1 -1835.761,E2 -1835.761} C_VEL
LIN {X 0,Y 580.277,Z 258.014,A -85,B 0,C 180,E1 -1838.147,E2 -1838.147} C_VEL
LIN {X 0,Y 580.288,Z 258.013,A -85,B 0,C 180,E1 -1840.844,E2 -1840.844} C_VEL
LIN {X 0,Y 580.259,Z 258.011,A -85,B 0,C 180,E1 -1843.66,E2 -1843.66} C_VEL
LIN {X 0,Y 580.266,Z 258.019,A -85,B 0,C 180,E1 -1846.61,E2 -1846.61} C_VEL
LIN {X 0,Y 580.282,Z 258.008,A -85,B 0,C 180,E1 -1849.731,E2 -1849.731} C_VEL
LIN {X 0,Y 580.29,Z 258.014,A -85,B 0,C 180,E1 -1852.732,E2 -1852.732} C_VEL
LIN {X 0,Y 580.284,Z 258.012,A -85,B 0,C 180,E1 -1855.443,E2 -1855.443} C_VEL
LIN {X 0,Y 580.293,Z 258.007,A -85,B 0,C 180,E1 -1857.971,E2 -1857.971} C_VEL
LIN {X 0,Y 580.283,Z 258.015,A -85,B 0,C 180,E1 -1861.024,E2 -1861.024} C_VEL
LIN {X 0,Y 580.26,Z 258.017,A -85,B 0,C 180,E1 -1863.672,E2 -1863.672} C_VEL
LIN {X 0,Y 580.256,Z 258.012,A -85,B 0,C 180,E1 -1866.442,E2 -1866.442} C_VEL
LIN {X 0,Y 580.307,Z 258.115,A -85,B 0,C 180,E1 -1868.417,E2 -1868.417} C_VEL
LIN {X 0,Y 580.651,Z 262.087,A -85,B 0,C 180,E1 -1869.108,E2 -1869.108} C_VEL
LIN {X 0,Y 580.491,Z 278.149,A -85,B 0,C 180,E1 -1871.836,E2 -1871.836} C_VEL
LIN {X 0,Y 580.407,Z 293.289,A -85,B 0,C 180,E1 -1874.371,E2 -1874.371} C_VEL
LIN {X 0,Y 580.29,Z 311.672,A -85,B 0,C 180,E1 -1877.409,E2 -1877.409} C_VEL
LIN {X 0,Y 580.215,Z 322.949,A -85,B 0,C 180,E1 -1879.255,E2 -1879.255} C_VEL
LIN {X 0,Y 580.617,Z 328.935,A -85,B 0,C 180,E1 -1879.341,E2 -1879.341} C_VEL
LIN {X 0,Y 580.536,Z 399.156,A -85,B 0,C 180,E1 -1880.22,E2 -1880.22} C_VEL
LIN {X 0,Y 580.479,Z 408.424,A -85,B 0,C 180,E1 -1880.417,E2 -1880.417} C_VEL
LIN {X 0,Y 580.446,Z 416.899,A -85,B 0,C 180,E1 -1880.681,E2 -1880.681} C_VEL
LIN {X 0,Y 580.4,Z 425.406,A -85,B 0,C 180,E1 -1881.031,E2 -1881.031} C_VEL
LIN {X 0,Y 580.381,Z 433.736,A -85,B 0,C 180,E1 -1881.47,E2 -1881.47} C_VEL
LIN {X 0,Y 580.284,Z 441.771,A -85,B 0,C 180,E1 -1881.994,E2 -1881.994} C_VEL
LIN {X 0,Y 580.222,Z 450.433,A -85,B 0,C 180,E1 -1882.693,E2 -1882.693} C_VEL
LIN {X 0,Y 580.204,Z 458.993,A -85,B 0,C 180,E1 -1883.574,E2 -1883.574} C_VEL
LIN {X 0,Y 580.15,Z 465.611,A -85,B 0,C 180,E1 -1884.439,E2 -1884.439} C_VEL
LIN {X 0,Y 580.096,Z 469.988,A -85,B 0,C 180,E1 -1885.135,E2 -1885.135} C_VEL
LIN {X 0,Y 580.137,Z 475.148,A -85,B 0,C 180,E1 -1886.18,E2 -1886.18} C_VEL
LIN {X 0,Y 580.07,Z 477.789,A -85,B 0,C 180,E1 -1886.875,E2 -1886.875} C_VEL
LIN {X 0,Y 580.04,Z 480.681,A -85,B 0,C 180,E1 -1887.917,E2 -1887.917} C_VEL
LIN {X 0,Y 580.045,Z 481.936,A -85,B 0,C 180,E1 -1888.611,E2 -1888.611} C_VEL
LIN {X 0,Y 580.036,Z 482.711,A -85,B 0,C 180,E1 -1889.306,E2 -1889.306} C_VEL
LIN {X 0,Y 580.034,Z 483,A -85,B 0,C 180,E1 -1890,E2 -1890} C_VEL
LIN {X 0,Y 580.036,Z 482.711,A -85,B 0,C 180,E1 -1890.694,E2 -1890.694} C_VEL
LIN {X 0,Y 580.045,Z 481.936,A -85,B 0,C 180,E1 -1891.389,E2 -1891.389} C_VEL
LIN {X 0,Y 580.04,Z 480.681,A -85,B 0,C 180,E1 -1892.083,E2 -1892.083} C_VEL
LIN {X 0,Y 580.07,Z 477.788,A -85,B 0,C 180,E1 -1893.125,E2 -1893.125} C_VEL
LIN {X 0,Y 580.137,Z 475.148,A -85,B 0,C 180,E1 -1893.82,E2 -1893.82} C_VEL
LIN {X 0,Y 580.096,Z 469.986,A -85,B 0,C 180,E1 -1894.865,E2 -1894.865} C_VEL
LIN {X 0,Y 580.193,Z 463.188,A -85,B 0,C 180,E1 -1895.91,E2 -1895.91} C_VEL
LIN {X 0,Y 580.225,Z 455.497,A -85,B 0,C 180,E1 -1896.808,E2 -1896.808} C_VEL
LIN {X 0,Y 580.249,Z 448.41,A -85,B 0,C 180,E1 -1897.481,E2 -1897.481} C_VEL
LIN {X 0,Y 580.303,Z 440.55,A -85,B 0,C 180,E1 -1898.093,E2 -1898.093} C_VEL
LIN {X 0,Y 580.428,Z 430.737,A -85,B 0,C 180,E1 -1898.705,E2 -1898.705} C_VEL
LIN {X 0,Y 580.421,Z 419.31,A -85,B 0,C 180,E1 -1899.232,E2 -1899.232} C_VEL
LIN {X 0,Y 580.477,Z 409.258,A -85,B 0,C 180,E1 -1899.561,E2 -1899.561} C_VEL
LIN {X 0,Y 580.526,Z 400.461,A -85,B 0,C 180,E1 -1899.758,E2 -1899.758} C_VEL
LIN {X 0,Y 580.607,Z 331.947,A -85,B 0,C 180,E1 -1900.622,E2 -1900.622} C_VEL
LIN {X 0,Y 580.302,Z 323.787,A -85,B 0,C 180,E1 -1900.728,E2 -1900.728} C_VEL
LIN {X 0,Y 580.218,Z 322.923,A -85,B 0,C 180,E1 -1900.75,E2 -1900.75} C_VEL
LIN {X 0,Y 580.311,Z 305.184,A -85,B 0,C 180,E1 -1903.66,E2 -1903.66} C_VEL
LIN {X 0,Y 580.477,Z 287.882,A -85,B 0,C 180,E1 -1906.53,E2 -1906.53} C_VEL
LIN {X 0,Y 580.586,Z 269.44,A -85,B 0,C 180,E1 -1909.637,E2 -1909.637} C_VEL
LIN {X 0,Y 580.524,Z 259.763,A -85,B 0,C 180,E1 -1911.295,E2 -1911.295} C_VEL
LIN {X 0,Y 580.291,Z 258.014,A -85,B 0,C 180,E1 -1911.631,E2 -1911.631} C_VEL
LIN {X 0,Y 580.264,Z 258.018,A -85,B 0,C 180,E1 -1914.317,E2 -1914.317} C_VEL
LIN {X 0,Y 580.249,Z 258.024,A -85,B 0,C 180,E1 -1916.624,E2 -1916.624} C_VEL
LIN {X 0,Y 580.273,Z 258.012,A -85,B 0,C 180,E1 -1919.305,E2 -1919.305} C_VEL
LIN {X 0,Y 580.288,Z 258.009,A -85,B 0,C 180,E1 -1922.2,E2 -1922.2} C_VEL
LIN {X 0,Y 580.279,Z 258.015,A -85,B 0,C 180,E1 -1924.696,E2 -1924.696} C_VEL
LIN {X 0,Y 580.289,Z 258.015,A -85,B 0,C 180,E1 -1927.268,E2 -1927.268} C_VEL
LIN {X 0,Y 580.282,Z 258.009,A -85,B 0,C 180,E1 -1930.269,E2 -1930.269} C_VEL
LIN {X 0,Y 580.266,Z 258.02,A -85,B 0,C 180,E1 -1933.39,E2 -1933.39} C_VEL
LIN {X 0,Y 580.258,Z 258.011,A -85,B 0,C 180,E1 -1936.34,E2 -1936.34} C_VEL
LIN {X 0,Y 580.288,Z 258.013,A -85,B 0,C 180,E1 -1939.156,E2 -1939.156} C_VEL
LIN {X 0,Y 580.279,Z 258.013,A -85,B 0,C 180,E1 -1941.926,E2 -1941.926} C_VEL
LIN {X 0,Y 580.27,Z 258.01,A -85,B 0,C 180,E1 -1944.454,E2 -1944.454} C_VEL
LIN {X 0,Y 580.277,Z 258.009,A -85,B 0,C 180,E1 -1946.974,E2 -1946.974} C_VEL
LIN {X 0,Y 580.289,Z 258.011,A -85,B 0,C 180,E1 -1949.425,E2 -1949.425} C_VEL
LIN {X 0,Y 580.284,Z 258.014,A -85,B 0,C 180,E1 -1952.141,E2 -1952.141} C_VEL
LIN {X 0,Y 580.307,Z 258.005,A -85,B 0,C 180,E1 -1955.269,E2 -1955.269} C_VEL
LIN {X 0,Y 580.256,Z 258.018,A -85,B 0,C 180,E1 -1957.947,E2 -1957.947} C_VEL
LIN {X 0,Y 580.283,Z 258.009,A -85,B 0,C 180,E1 -1960.913,E2 -1960.913} C_VEL
LIN {X 0,Y 580.253,Z 258.014,A -85,B 0,C 180,E1 -1963.825,E2 -1963.825} C_VEL
LIN {X 0,Y 580.258,Z 258.018,A -85,B 0,C 180,E1 -1966.696,E2 -1966.696} C_VEL
LIN {X 0,Y 580.295,Z 258.006,A -85,B 0,C 180,E1 -1969.533,E2 -1969.533} C_VEL
LIN {X 0,Y 580.312,Z 258.009,A -85,B 0,C 180,E1 -1972.345,E2 -1972.345} C_VEL
LIN {X 0,Y 580.332,Z 258.006,A -85,B 0,C 180,E1 -1975.137,E2 -1975.137} C_VEL
LIN {X 0,Y 580.312,Z 258.004,A -85,B 0,C 180,E1 -1977.918,E2 -1977.918} C_VEL
LIN {X 0,Y 580.346,Z 258.006,A -85,B 0,C 180,E1 -1980.694,E2 -1980.694} C_VEL
LIN {X 0,Y 580.283,Z 258.012,A -85,B 0,C 180,E1 -1983.472,E2 -1983.472} C_VEL
LIN {X 0,Y 580.322,Z 258.007,A -85,B 0,C 180,E1 -1985.56,E2 -1985.56} C_VEL
LIN {X 0,Y 580.314,Z 258.004,A -85,B 0,C 180,E1 -1988.356,E2 -1988.356} C_VEL
LIN {X 0,Y 580.285,Z 258.016,A -85,B 0,C 180,E1 -1991.191,E2 -1991.191} C_VEL
LIN {X 0,Y 580.313,Z 258.007,A -85,B 0,C 180,E1 -1994.017,E2 -1994.017} C_VEL
LIN {X 0,Y 580.298,Z 258.007,A -85,B 0,C 180,E1 -1996.914,E2 -1996.914} C_VEL
LIN {X 0,Y 580.292,Z 258.015,A -85,B 0,C 180,E1 -1999.823,E2 -1999.823} C_VEL
LIN {X 0,Y 580.27,Z 258.014,A -85,B 0,C 180,E1 -2001.316,E2 -2001.316} C_VEL
LIN {X 0,Y 579.573,Z 258.105,A -85,B 0,C 180,E1 -2001.895,E2 -2001.895} C_VEL
LIN {X 0,Y 576.698,Z 258.461,A -85,B 0,C 180,E1 -2002.835,E2 -2002.835} C_VEL
LIN {X 0,Y 574.304,Z 258.761,A -85,B 0,C 180,E1 -2003.591,E2 -2003.591} C_VEL
LIN {X 0,Y 573.304,Z 258.883,A -85,B 0,C 180,E1 -2004.175,E2 -2004.175} C_VEL
LIN {X 0,Y 573.237,Z 258.889,A -85,B 0,C 180,E1 -2004.373,E2 -2004.373} C_VEL
LIN {X 0,Y 573.252,Z 258.884,A -85,B 0,C 180,E1 -2006.976,E2 -2006.976} C_VEL
LIN {X 0,Y 573.241,Z 258.888,A -85,B 0,C 180,E1 -2009.49,E2 -2009.49} C_VEL
LIN {X 0,Y 573.243,Z 258.888,A -85,B 0,C 180,E1 -2012.646,E2 -2012.646} C_VEL
LIN {X 0,Y 573.259,Z 258.883,A -85,B 0,C 180,E1 -2015.184,E2 -2015.184} C_VEL
LIN {X 0,Y 573.227,Z 258.891,A -85,B 0,C 180,E1 -2017.808,E2 -2017.808} C_VEL
LIN {X 0,Y 573.261,Z 258.893,A -85,B 0,C 180,E1 -2020.529,E2 -2020.529} C_VEL
LIN {X 0,Y 573.29,Z 258.929,A -85,B 0,C 180,E1 -2023.791,E2 -2023.791} C_VEL
LIN {X 0,Y 573.281,Z 270.954,A -85,B 0,C 180,E1 -2026.327,E2 -2026.327} C_VEL
LIN {X 0,Y 573.177,Z 284.955,A -85,B 0,C 180,E1 -2029.239,E2 -2029.239} C_VEL
LIN {X 0,Y 573.16,Z 294.657,A -85,B 0,C 180,E1 -2031.193,E2 -2031.193} C_VEL
LIN {X 0,Y 573.614,Z 300.431,A -85,B 0,C 180,E1 -2031.273,E2 -2031.273} C_VEL
LIN {X 0,Y 573.534,Z 370.453,A -85,B 0,C 180,E1 -2032.167,E2 -2032.167} C_VEL
LIN {X 0,Y 573.501,Z 380.618,A -85,B 0,C 180,E1 -2032.403,E2 -2032.403} C_VEL
LIN {X 0,Y 573.417,Z 392.171,A -85,B 0,C 180,E1 -2032.813,E2 -2032.813} C_VEL
LIN {X 0,Y 573.363,Z 401.995,A -85,B 0,C 180,E1 -2033.306,E2 -2033.306} C_VEL
LIN {X 0,Y 573.257,Z 410.444,A -85,B 0,C 180,E1 -2033.844,E2 -2033.844} C_VEL
LIN {X 0,Y 573.164,Z 418.598,A -85,B 0,C 180,E1 -2034.487,E2 -2034.487} C_VEL
LIN {X 0,Y 573.135,Z 424.52,A -85,B 0,C 180,E1 -2035.051,E2 -2035.051} C_VEL
LIN {X 0,Y 573.097,Z 429.977,A -85,B 0,C 180,E1 -2035.661,E2 -2035.661} C_VEL
LIN {X 0,Y 573.074,Z 434.811,A -85,B 0,C 180,E1 -2036.295,E2 -2036.295} C_VEL
LIN {X 0,Y 573.054,Z 440.072,A -85,B 0,C 180,E1 -2037.136,E2 -2037.136} C_VEL
LIN {X 0,Y 573.001,Z 443.576,A -85,B 0,C 180,E1 -2037.812,E2 -2037.812} C_VEL
LIN {X 0,Y 573,Z 446.813,A -85,B 0,C 180,E1 -2038.583,E2 -2038.583} C_VEL
LIN {X 0,Y 572.955,Z 450.389,A -85,B 0,C 180,E1 -2039.808,E2 -2039.808} C_VEL
LIN {X 0,Y 572.981,Z 451.906,A -85,B 0,C 180,E1 -2040.619,E2 -2040.619} C_VEL
LIN {X 0,Y 572.93,Z 452.745,A -85,B 0,C 180,E1 -2041.42,E2 -2041.42} C_VEL
LIN {X 0,Y 572.947,Z 452.948,A -85,B 0,C 180,E1 -2042.218,E2 -2042.218} C_VEL
LIN {X 0,Y 572.933,Z 452.525,A -85,B 0,C 180,E1 -2043.009,E2 -2043.009} C_VEL
LIN {X 0,Y 572.942,Z 451.453,A -85,B 0,C 180,E1 -2043.795,E2 -2043.795} C_VEL
LIN {X 0,Y 572.958,Z 449.712,A -85,B 0,C 180,E1 -2044.577,E2 -2044.577} C_VEL
LIN {X 0,Y 572.988,Z 445.894,A -85,B 0,C 180,E1 -2045.74,E2 -2045.74} C_VEL
LIN {X 0,Y 573.025,Z 441.446,A -85,B 0,C 180,E1 -2046.701,E2 -2046.701} C_VEL
LIN {X 0,Y 573.068,Z 436.988,A -85,B 0,C 180,E1 -2047.468,E2 -2047.468} C_VEL
LIN {X 0,Y 573.096,Z 431.611,A -85,B 0,C 180,E1 -2048.226,E2 -2048.226} C_VEL
LIN {X 0,Y 573.135,Z 425.321,A -85,B 0,C 180,E1 -2048.956,E2 -2048.956} C_VEL
LIN {X 0,Y 573.2,Z 418.141,A -85,B 0,C 180,E1 -2049.641,E2 -2049.641} C_VEL
LIN {X 0,Y 573.252,Z 411.018,A -85,B 0,C 180,E1 -2050.204,E2 -2050.204} C_VEL
LIN {X 0,Y 573.348,Z 403.255,A -85,B 0,C 180,E1 -2050.709,E2 -2050.709} C_VEL
LIN {X 0,Y 573.393,Z 395.017,A -85,B 0,C 180,E1 -2051.143,E2 -2051.143} C_VEL
LIN {X 0,Y 573.441,Z 386.014,A -85,B 0,C 180,E1 -2051.512,E2 -2051.512} C_VEL
LIN {X 0,Y 573.533,Z 375.358,A -85,B 0,C 180,E1 -2051.827,E2 -2051.827} C_VEL
LIN {X 0,Y 573.566,Z 360.357,A -85,B 0,C 180,E1 -2052.07,E2 -2052.07} C_VEL
LIN {X 0,Y 573.575,Z 297.593,A -85,B 0,C 180,E1 -2052.853,E2 -2052.853} C_VEL
LIN {X 0,Y 573.117,Z 294.32,A -85,B 0,C 180,E1 -2052.922,E2 -2052.922} C_VEL
LIN {X 0,Y 573.188,Z 280.349,A -85,B 0,C 180,E1 -2055.805,E2 -2055.805} C_VEL
LIN {X 0,Y 573.287,Z 266.327,A -85,B 0,C 180,E1 -2058.734,E2 -2058.734} C_VEL
LIN {X 0,Y 573.298,Z 258.882,A -85,B 0,C 180,E1 -2060.341,E2 -2060.341} C_VEL
LIN {X 0,Y 573.312,Z 258.88,A -85,B 0,C 180,E1 -2063.192,E2 -2063.192} C_VEL
LIN {X 0,Y 573.223,Z 258.899,A -85,B 0,C 180,E1 -2065.781,E2 -2065.781} C_VEL
LIN {X 0,Y 573.307,Z 258.887,A -85,B 0,C 180,E1 -2067.892,E2 -2067.892} C_VEL
LIN {X 0,Y 573.328,Z 258.875,A -85,B 0,C 180,E1 -2070.702,E2 -2070.702} C_VEL
LIN {X 0,Y 573.302,Z 258.878,A -85,B 0,C 180,E1 -2072.811,E2 -2072.811} C_VEL
LIN {X 0,Y 573.289,Z 258.882,A -85,B 0,C 180,E1 -2075.628,E2 -2075.628} C_VEL
LIN {X 0,Y 573.283,Z 258.887,A -85,B 0,C 180,E1 -2078.459,E2 -2078.459} C_VEL
LIN {X 0,Y 573.274,Z 258.881,A -85,B 0,C 180,E1 -2081.312,E2 -2081.312} C_VEL
LIN {X 0,Y 573.283,Z 258.892,A -85,B 0,C 180,E1 -2084.424,E2 -2084.424} C_VEL
LIN {X 0,Y 573.259,Z 258.885,A -85,B 0,C 180,E1 -2087.111,E2 -2087.111} C_VEL
LIN {X 0,Y 573.242,Z 258.887,A -85,B 0,C 180,E1 -2090.076,E2 -2090.076} C_VEL
LIN {X 0,Y 573.233,Z 258.891,A -85,B 0,C 180,E1 -2092.337,E2 -2092.337} C_VEL
LIN {X 0,Y 573.245,Z 258.887,A -85,B 0,C 180,E1 -2095.41,E2 -2095.41} C_VEL
LIN {X 0,Y 573.25,Z 258.884,A -85,B 0,C 180,E1 -2098.028,E2 -2098.028} C_VEL
LIN {X 0,Y 573.227,Z 258.896,A -85,B 0,C 180,E1 -2100.882,E2 -2100.882} C_VEL
LIN {X 0,Y 573.237,Z 258.89,A -85,B 0,C 180,E1 -2103.52,E2 -2103.52} C_VEL
LIN {X 0,Y 573.21,Z 258.889,A -85,B 0,C 180,E1 -2106.051,E2 -2106.051} C_VEL
LIN {X 0,Y 573.236,Z 258.888,A -85,B 0,C 180,E1 -2108.701,E2 -2108.701} C_VEL
LIN {X 0,Y 573.225,Z 258.895,A -85,B 0,C 180,E1 -2111.592,E2 -2111.592} C_VEL
LIN {X 0,Y 573.228,Z 258.887,A -85,B 0,C 180,E1 -2114.332,E2 -2114.332} C_VEL
LIN {X 0,Y 573.243,Z 258.892,A -85,B 0,C 180,E1 -2117.356,E2 -2117.356} C_VEL
LIN {X 0,Y 573.24,Z 258.886,A -85,B 0,C 180,E1 -2120.392,E2 -2120.392} C_VEL
LIN {X 0,Y 573.248,Z 258.885,A -85,B 0,C 180,E1 -2123.077,E2 -2123.077} C_VEL
LIN {X 0,Y 573.265,Z 258.889,A -85,B 0,C 180,E1 -2125.671,E2 -2125.671} C_VEL
LIN {X 0,Y 573.231,Z 258.894,A -85,B 0,C 180,E1 -2128.184,E2 -2128.184} C_VEL
LIN {X 0,Y 573.258,Z 258.885,A -85,B 0,C 180,E1 -2130.634,E2 -2130.634} C_VEL
LIN {X 0,Y 573.258,Z 258.884,A -85,B 0,C 180,E1 -2133.5,E2 -2133.5} C_VEL
LIN {X 0,Y 573.222,Z 258.896,A -85,B 0,C 180,E1 -2136.134,E2 -2136.134} C_VEL
LIN {X 0,Y 573.238,Z 258.886,A -85,B 0,C 180,E1 -2139.173,E2 -2139.173} C_VEL
LIN {X 0,Y 573.217,Z 258.888,A -85,B 0,C 180,E1 -2141.411,E2 -2141.411} C_VEL
LIN {X 0,Y 573.241,Z 258.885,A -85,B 0,C 180,E1 -2143.621,E2 -2143.621} C_VEL
LIN {X 0,Y 573.26,Z 258.883,A -85,B 0,C 180,E1 -2145.807,E2 -2145.807} C_VEL
LIN {X 0,Y 573.248,Z 258.895,A -85,B 0,C 180,E1 -2148.745,E2 -2148.745} C_VEL
LIN {X 0,Y 573.271,Z 258.882,A -85,B 0,C 180,E1 -2151.54,E2 -2151.54} C_VEL
LIN {X 0,Y 573.289,Z 258.882,A -85,B 0,C 180,E1 -2154.372,E2 -2154.372} C_VEL
LIN {X 0,Y 573.291,Z 258.887,A -85,B 0,C 180,E1 -2157.189,E2 -2157.189} C_VEL
LIN {X 0,Y 573.298,Z 258.878,A -85,B 0,C 180,E1 -2160,E2 -2160} C_VEL
LIN {X 0,Y 573.303,Z 258.882,A -85,B 0,C 180,E1 -2162.811,E2 -2162.811} C_VEL
LIN {X 0,Y 573.28,Z 258.886,A -85,B 0,C 180,E1 -2165.628,E2 -2165.628} C_VEL
LIN {X 0,Y 573.262,Z 258.883,A -85,B 0,C 180,E1 -2168.46,E2 -2168.46} C_VEL
LIN {X 0,Y 573.286,Z 258.887,A -85,B 0,C 180,E1 -2171.312,E2 -2171.312} C_VEL
LIN {X 0,Y 573.266,Z 258.882,A -85,B 0,C 180,E1 -2174.425,E2 -2174.425} C_VEL
LIN {X 0,Y 573.245,Z 258.887,A -85,B 0,C 180,E1 -2177.112,E2 -2177.112} C_VEL
LIN {X 0,Y 573.236,Z 258.892,A -85,B 0,C 180,E1 -2180.077,E2 -2180.077} C_VEL
LIN {X 0,Y 573.221,Z 258.888,A -85,B 0,C 180,E1 -2183.1,E2 -2183.1} C_VEL
LIN {X 0,Y 573.244,Z 258.887,A -85,B 0,C 180,E1 -2185.41,E2 -2185.41} C_VEL
LIN {X 0,Y 573.222,Z 258.891,A -85,B 0,C 180,E1 -2188.565,E2 -2188.565} C_VEL
LIN {X 0,Y 573.216,Z 258.889,A -85,B 0,C 180,E1 -2190.994,E2 -2190.994} C_VEL
LIN {X 0,Y 573.251,Z 258.885,A -85,B 0,C 180,E1 -2193.525,E2 -2193.525} C_VEL
LIN {X 0,Y 573.233,Z 258.891,A -85,B 0,C 180,E1 -2196.05,E2 -2196.05} C_VEL
LIN {X 0,Y 573.229,Z 258.894,A -85,B 0,C 180,E1 -2198.703,E2 -2198.703} C_VEL
LIN {X 0,Y 573.232,Z 258.886,A -85,B 0,C 180,E1 -2201.595,E2 -2201.595} C_VEL
LIN {X 0,Y 573.219,Z 258.893,A -85,B 0,C 180,E1 -2204.335,E2 -2204.335} C_VEL
LIN {X 0,Y 573.218,Z 258.89,A -85,B 0,C 180,E1 -2207.361,E2 -2207.361} C_VEL
LIN {X 0,Y 573.234,Z 258.889,A -85,B 0,C 180,E1 -2210.393,E2 -2210.393} C_VEL
LIN {X 0,Y 573.245,Z 258.894,A -85,B 0,C 180,E1 -2213.078,E2 -2213.078} C_VEL
LIN {X 0,Y 573.248,Z 258.886,A -85,B 0,C 180,E1 -2215.671,E2 -2215.671} C_VEL
LIN {X 0,Y 573.23,Z 258.887,A -85,B 0,C 180,E1 -2218.185,E2 -2218.185} C_VEL
LIN {X 0,Y 573.237,Z 258.887,A -85,B 0,C 180,E1 -2220.634,E2 -2220.634} C_VEL
LIN {X 0,Y 573.208,Z 258.898,A -85,B 0,C 180,E1 -2223.513,E2 -2223.513} C_VEL
LIN {X 0,Y 573.206,Z 258.892,A -85,B 0,C 180,E1 -2226.134,E2 -2226.134} C_VEL
LIN {X 0,Y 573.278,Z 259.06,A -85,B 0,C 180,E1 -2228.328,E2 -2228.328} C_VEL
LIN {X 0,Y 573.645,Z 263.995,A -85,B 0,C 180,E1 -2229.189,E2 -2229.189} C_VEL
LIN {X 0,Y 573.487,Z 279.23,A -85,B 0,C 180,E1 -2231.791,E2 -2231.791} C_VEL
LIN {X 0,Y 573.398,Z 294.37,A -85,B 0,C 180,E1 -2234.357,E2 -2234.357} C_VEL
LIN {X 0,Y 573.244,Z 311.672,A -85,B 0,C 180,E1 -2237.251,E2 -2237.251} C_VEL
LIN {X 0,Y 573.171,Z 322.969,A -85,B 0,C 180,E1 -2239.124,E2 -2239.124} C_VEL
LIN {X 0,Y 573.661,Z 329.712,A -85,B 0,C 180,E1 -2239.22,E2 -2239.22} C_VEL
LIN {X 0,Y 573.544,Z 399.156,A -85,B 0,C 180,E1 -2240.1,E2 -2240.1} C_VEL
LIN {X 0,Y 573.472,Z 408.423,A -85,B 0,C 180,E1 -2240.299,E2 -2240.299} C_VEL
LIN {X 0,Y 573.443,Z 416.897,A -85,B 0,C 180,E1 -2240.566,E2 -2240.566} C_VEL
LIN {X 0,Y 573.39,Z 425.403,A -85,B 0,C 180,E1 -2240.921,E2 -2240.921} C_VEL
LIN {X 0,Y 573.366,Z 433.734,A -85,B 0,C 180,E1 -2241.364,E2 -2241.364} C_VEL
LIN {X 0,Y 573.256,Z 441.773,A -85,B 0,C 180,E1 -2241.895,E2 -2241.895} C_VEL
LIN {X 0,Y 573.175,Z 450.433,A -85,B 0,C 180,E1 -2242.603,E2 -2242.603} C_VEL
LIN {X 0,Y 573.154,Z 458.464,A -85,B 0,C 180,E1 -2243.429,E2 -2243.429} C_VEL
LIN {X 0,Y 573.112,Z 464.435,A -85,B 0,C 180,E1 -2244.194,E2 -2244.194} C_VEL
LIN {X 0,Y 573.004,Z 469.989,A -85,B 0,C 180,E1 -2245.075,E2 -2245.075} C_VEL
LIN {X 0,Y 573.036,Z 475.149,A -85,B 0,C 180,E1 -2246.132,E2 -2246.132} C_VEL
LIN {X 0,Y 572.99,Z 477.788,A -85,B 0,C 180,E1 -2246.836,E2 -2246.836} C_VEL
LIN {X 0,Y 572.94,Z 480.682,A -85,B 0,C 180,E1 -2247.891,E2 -2247.891} C_VEL
LIN {X 0,Y 572.944,Z 481.934,A -85,B 0,C 180,E1 -2248.594,E2 -2248.594} C_VEL
